# B&R Automation Studio project NAELD004C00R10L518F00 (part 2)

### IoMap.iom - X20CP0483/IoMap.iom
```iecst
VAR_CONFIG
	::DInput:a_bPhysicalDI[1] AT %IX."X20DI9372".DigitalInput01;
	::DInput:a_bPhysicalDI[2] AT %IX."X20DI9372".DigitalInput02;
	::DInput:a_bPhysicalDI[3] AT %IX."X20DI9372".DigitalInput03;
	::DInput:a_bPhysicalDI[4] AT %IX."X20DI9372".DigitalInput04;
	::DInput:a_bPhysicalDI[5] AT %IX."X20DI9372".DigitalInput05;
	::DInput:a_bPhysicalDI[6] AT %IX."X20DI9372".DigitalInput06;
	::DInput:a_bPhysicalDI[7] AT %IX."X20DI9372".DigitalInput07;
	::DInput:a_bPhysicalDI[8] AT %IX."X20DI9372".DigitalInput08;
	::DInput:a_bPhysicalDI[9] AT %IX."X20DI9372".DigitalInput09;
	::DInput:a_bPhysicalDI[10] AT %IX."X20DI9372".DigitalInput10;
	::DInput:a_bPhysicalDI[11] AT %IX."X20DI9372".DigitalInput11;
	::DInput:a_bPhysicalDI[12] AT %IX."X20DI9372".DigitalInput12;
	::DInput:a_bPhysicalDI[13] AT %IX."X20DI9372a".DigitalInput01;
	::DInput:a_bPhysicalDI[14] AT %IX."X20DI9372a".DigitalInput02;
	::DInput:a_bPhysicalDI[15] AT %IX."X20DI9372a".DigitalInput03;
	::DInput:a_bPhysicalDI[16] AT %IX."X20DI9372a".DigitalInput04;
	::DInput:a_bPhysicalDI[17] AT %IX."X20DI9372a".DigitalInput05;
	::DInput:a_bPhysicalDI[18] AT %IX."X20DI9372a".DigitalInput06;
	::DInput:a_bPhysicalDI[19] AT %IX."X20DI9372a".DigitalInput07;
	::DInput:a_bPhysicalDI[20] AT %IX."X20DI9372a".DigitalInput08;
	::DInput:a_bPhysicalDI[21] AT %IX."X20DI9372a".DigitalInput09;
	::DInput:a_bPhysicalDI[22] AT %IX."X20DI9372a".DigitalInput10;
	::DInput:a_bPhysicalDI[23] AT %IX."X20DI9372a".DigitalInput11;
	::DInput:a_bPhysicalDI[24] AT %IX."X20DI9372a".DigitalInput12;
	::DInput:a_bPhysicalDI[25] AT %IX."X20DI9372b".DigitalInput01;
	::DInput:a_bPhysicalDI[26] AT %IX."X20DI9372b".DigitalInput02;
	::DInput:a_bPhysicalDI[27] AT %IX."X20DI9372b".DigitalInput03;
	::DInput:a_bPhysicalDI[28] AT %IX."X20DI9372b".DigitalInput04;
	::DInput:a_bPhysicalDI[29] AT %IX."X20DI9372b".DigitalInput05;
	::DInput:a_bPhysicalDI[30] AT %IX."X20DI9372b".DigitalInput06;
	::DInput:a_bPhysicalDI[31] AT %IX."X20DI9372b".DigitalInput07;
	::DInput:a_bPhysicalDI[32] AT %IX."X20DI9372b".DigitalInput08;
	::DInput:a_bPhysicalDI[33] AT %IX."X20DI9372b".DigitalInput09;
	::DInput:a_bPhysicalDI[34] AT %IX."X20DI9372b".DigitalInput10;
	::DInput:a_bPhysicalDI[35] AT %IX."X20DI9372b".DigitalInput11;
	::DInput:a_bPhysicalDI[36] AT %IX."X20DI9372b".DigitalInput12;
	::DInput:a_bPhysicalDI[37] AT %IX."X20DI9372c".DigitalInput01;
	::DInput:a_bPhysicalDI[38] AT %IX."X20DI9372c".DigitalInput02;
	::DInput:a_bPhysicalDI[39] AT %IX."X20DI9372c".DigitalInput03;
	::DInput:a_bPhysicalDI[40] AT %IX."X20DI9372c".DigitalInput04;
	::DInput:a_bPhysicalDI[41] AT %IX."X20DI9372c".DigitalInput05;
	::DInput:a_bPhysicalDI[42] AT %IX."X20DI9372c".DigitalInput06;
	::DInput:a_bPhysicalDI[43] AT %IX."X20DI9372c".DigitalInput07;
	::DInput:a_bPhysicalDI[44] AT %IX."X20DI9372c".DigitalInput08;
	::DInput:a_bPhysicalDI[45] AT %IX."X20DI9372c".DigitalInput09;
	::DInput:a_bPhysicalDI[46] AT %IX."X20DI9372c".DigitalInput10;
	::DInput:a_bPhysicalDI[47] AT %IX."X20DI9372c".DigitalInput11;
	::DInput:a_bPhysicalDI[48] AT %IX."X20DI9372c".DigitalInput12;
	::DInput:a_bPhysicalDI[49] AT %IX."X20DI9372d".DigitalInput01;
	::DInput:a_bPhysicalDI[50] AT %IX."X20DI9372d".DigitalInput02;
	::DInput:a_bPhysicalDI[51] AT %IX."X20DI9372d".DigitalInput03;
	::DInput:a_bPhysicalDI[52] AT %IX."X20DI9372d".DigitalInput04;
	::DInput:a_bPhysicalDI[53] AT %IX."X20DI9372d".DigitalInput05;
	::DInput:a_bPhysicalDI[54] AT %IX."X20DI9372d".DigitalInput06;
	::DInput:a_bPhysicalDI[55] AT %IX."X20DI9372d".DigitalInput07;
	::DInput:a_bPhysicalDI[56] AT %IX."X20DI9372d".DigitalInput08;
	::DInput:a_bPhysicalDI[57] AT %IX."X20DI9372d".DigitalInput09;
	::DInput:a_bPhysicalDI[58] AT %IX."X20DI9372d".DigitalInput10;
	::DInput:a_bPhysicalDI[59] AT %IX."X20DI9372d".DigitalInput11;
	::DInput:a_bPhysicalDI[60] AT %IX."X20DI9372d".DigitalInput12;
	::DInput:a_bPhysicalDI[61] AT %IX."X20DI9372e".DigitalInput01;
	::DInput:a_bPhysicalDI[62] AT %IX."X20DI9372e".DigitalInput02;
	::DInput:a_bPhysicalDI[63] AT %IX."X20DI9372e".DigitalInput03;
	::DInput:a_bPhysicalDI[64] AT %IX."X20DI9372e".DigitalInput04;
	::DInput:a_bPhysicalDI[65] AT %IX."X20DI9372e".DigitalInput05;
	::DInput:a_bPhysicalDI[66] AT %IX."X20DI9372e".DigitalInput06;
	::DInput:a_bPhysicalDI[67] AT %IX."X20DI9372e".DigitalInput07;
	::DInput:a_bPhysicalDI[68] AT %IX."X20DI9372e".DigitalInput08;
	::DInput:a_bPhysicalDI[69] AT %IX."X20DI9372e".DigitalInput09;
	::DInput:a_bPhysicalDI[70] AT %IX."X20DI9372e".DigitalInput10;
	::DInput:a_bPhysicalDI[71] AT %IX."X20DI9372e".DigitalInput11;
	::DInput:a_bPhysicalDI[72] AT %IX."X20DI9372e".DigitalInput12;
	::DOutput:a_bPhysicalDO[1] AT %QX."X20DO6321".DigitalOutput01;
	::DOutput:a_bPhysicalDO[2] AT %QX."X20DO6321".DigitalOutput02;
	::DOutput:a_bPhysicalDO[3] AT %QX."X20DO6321".DigitalOutput03;
	::DOutput:a_bPhysicalDO[4] AT %QX."X20DO6321".DigitalOutput04;
	::DOutput:a_bPhysicalDO[5] AT %QX."X20DO6321".DigitalOutput05;
	::DOutput:a_bPhysicalDO[6] AT %QX."X20DO6321".DigitalOutput06;
	::DOutput:a_bPhysicalDO[7] AT %QX."X20DO9321".DigitalOutput01;
	::DOutput:a_bPhysicalDO[8] AT %QX."X20DO9321".DigitalOutput02;
	::DOutput:a_bPhysicalDO[9] AT %QX."X20DO9321".DigitalOutput03;
	::DOutput:a_bPhysicalDO[10] AT %QX."X20DO9321".DigitalOutput04;
	::DOutput:a_bPhysicalDO[11] AT %QX."X20DO9321".DigitalOutput05;
	::DOutput:a_bPhysicalDO[12] AT %QX."X20DO9321".DigitalOutput06;
	::DOutput:a_bPhysicalDO[13] AT %QX."X20DO9321".DigitalOutput07;
	::DOutput:a_bPhysicalDO[14] AT %QX."X20DO9321".DigitalOutput08;
	::DOutput:a_bPhysicalDO[15] AT %QX."X20DO9321".DigitalOutput09;
	::DOutput:a_bPhysicalDO[16] AT %QX."X20DO9321".DigitalOutput10;
	::DOutput:a_bPhysicalDO[17] AT %QX."X20DO9321".DigitalOutput11;
	::DOutput:a_bPhysicalDO[18] AT %QX."X20DO9321".DigitalOutput12;
	::DOutput:a_bPhysicalDO[19] AT %QX."X20DO9321a".DigitalOutput01;
	::DOutput:a_bPhysicalDO[20] AT %QX."X20DO9321a".DigitalOutput02;
	::DOutput:a_bPhysicalDO[21] AT %QX."X20DO9321a".DigitalOutput03;
	::DOutput:a_bPhysicalDO[22] AT %QX."X20DO9321a".DigitalOutput04;
	::DOutput:a_bPhysicalDO[23] AT %QX."X20DO9321a".DigitalOutput05;
	::DOutput:a_bPhysicalDO[24] AT %QX."X20DO9321a".DigitalOutput06;
	::DOutput:a_bPhysicalDO[25] AT %QX."X20DO9321a".DigitalOutput07;
	::DOutput:a_bPhysicalDO[26] AT %QX."X20DO9321a".DigitalOutput08;
	::DOutput:a_bPhysicalDO[27] AT %QX."X20DO9321a".DigitalOutput09;
	::DOutput:a_bPhysicalDO[28] AT %QX."X20DO9321a".DigitalOutput10;
	::DOutput:a_bPhysicalDO[29] AT %QX."X20DO9321a".DigitalOutput11;
	::DOutput:a_bPhysicalDO[30] AT %QX."X20DO9321a".DigitalOutput12;
	::DOutput:a_bPhysicalDO[31] AT %QX."X20DO9321b".DigitalOutput01;
	::DOutput:a_bPhysicalDO[32] AT %QX."X20DO9321b".DigitalOutput02;
	::DOutput:a_bPhysicalDO[33] AT %QX."X20DO9321b".DigitalOutput03;
	::DOutput:a_bPhysicalDO[34] AT %QX."X20DO9321b".DigitalOutput04;
	::DOutput:a_bPhysicalDO[35] AT %QX."X20DO9321b".DigitalOutput05;
	::DOutput:a_bPhysicalDO[36] AT %QX."X20DO9321b".DigitalOutput06;
	::DOutput:a_bPhysicalDO[37] AT %QX."X20DO9321b".DigitalOutput07;
	::DOutput:a_bPhysicalDO[38] AT %QX."X20DO9321b".DigitalOutput08;
	::DOutput:a_bPhysicalDO[39] AT %QX."X20DO9321b".DigitalOutput09;
	::DOutput:a_bPhysicalDO[40] AT %QX."X20DO9321b".DigitalOutput10;
	::DOutput:a_bPhysicalDO[41] AT %QX."X20DO9321b".DigitalOutput11;
	::DOutput:a_bPhysicalDO[42] AT %QX."X20DO9321b".DigitalOutput12;
	::DOutput:a_bPhysicalDO[43] AT %QX."X20DO9321c".DigitalOutput01;
	::DOutput:a_bPhysicalDO[44] AT %QX."X20DO9321c".DigitalOutput02;
	::DOutput:a_bPhysicalDO[45] AT %QX."X20DO9321c".DigitalOutput03;
	::DOutput:a_bPhysicalDO[46] AT %QX."X20DO9321c".DigitalOutput04;
	::DOutput:a_bPhysicalDO[47] AT %QX."X20DO9321c".DigitalOutput05;
	::DOutput:a_bPhysicalDO[48] AT %QX."X20DO9321c".DigitalOutput06;
	::DOutput:a_bPhysicalDO[49] AT %QX."X20DO9321c".DigitalOutput07;
	::DOutput:a_bPhysicalDO[50] AT %QX."X20DO9321c".DigitalOutput08;
	::DOutput:a_bPhysicalDO[51] AT %QX."X20DO9321c".DigitalOutput09;
	::DOutput:a_bPhysicalDO[52] AT %QX."X20DO9321c".DigitalOutput10;
	::DOutput:a_bPhysicalDO[53] AT %QX."X20DO9321c".DigitalOutput11;
	::DOutput:a_bPhysicalDO[54] AT %QX."X20DO9321c".DigitalOutput12;
	::LifterBtm:bModuleOK AT %IX."Lifter".ModuleOk;
	::LifterBtm:tyParamInDriver.uiErrCode_603F AT %IW."Lifter".ErrorCode_603F;
	::LifterBtm:tyParamOutDriver.uiCtrlword_6040 AT %QW."Lifter".Controlword_6040;
	::LifterBtm:tyParamInDriver.uiStatword_6041 AT %IW."Lifter".Statusword_6041;
	::LifterBtm:tyParamOutDriver.siModOfOpt_6060 AT %QB."Lifter".ModesOfOperation_6060;
	::LifterBtm:tyParamInDriver.siModOfOptDisp_6061 AT %IB."Lifter".ModesOfOperationDisplay_6061;
	::LifterBtm:tyParamInDriver.diActualPos_6064 AT %ID."Lifter".PositionActualValue_6064;
	::LifterBtm:tyParamOutDriver.diTargetPos_607A AT %QD."Lifter".TargetPosition_607A;
	::LifterBtm:tyParamOutDriver.udiMoveSpd_6081 AT %QD."Lifter".ProfileVelocity_6081;
	::LifterBtm:tyParamOutDriver.siHmMethod_6098 AT %QB."Lifter".HomingMethod_6098;
	::LifterBtm:tyParamInDriver.udiDigitalInputs_60FD AT %ID."Lifter".DigitalInputs_60FD;
	::LifterBtm:tyParamOutDriver.diJogVel_60FF AT %QD."Lifter".TargetVelocity_60FF;
	::Trav:bModuleOK AT %IX."Traverser".ModuleOk;
	::Trav:tyParamInDriver.uiErrCode_603F AT %IW."Traverser".ErrorCode_603F;
	::Trav:tyParamOutDriver.uiCtrlword_6040 AT %QW."Traverser".Controlword_6040;
	::Trav:tyParamInDriver.uiStatword_6041 AT %IW."Traverser".Statusword_6041;
	::Trav:tyParamOutDriver.siModOfOpt_6060 AT %QB."Traverser".ModesOfOperation_6060;
	::Trav:tyParamInDriver.siModOfOptDisp_6061 AT %IB."Traverser".ModesOfOperationDisplay_6061;
	::Trav:tyParamInDriver.diActualPos_6064 AT %ID."Traverser".PositionActualValue_6064;
	::Trav:tyParamOutDriver.diTargetPos_607A AT %QD."Traverser".TargetPosition_607A;
	::Trav:tyParamOutDriver.udiMoveSpd_6081 AT %QD."Traverser".ProfileVelocity_6081;
	::Trav:tyParamOutDriver.siHmMethod_6098 AT %QB."Traverser".HomingMethod_6098;
	::Trav:tyParamInDriver.udiDigitalInputs_60FD AT %ID."Traverser".DigitalInputs_60FD;
	::Trav:tyParamOutDriver.diJogVel_60FF AT %QD."Traverser".TargetVelocity_60FF;
	::AWOpen:bModuleOK AT %IX."AutoWidthConv".ModuleOk;
	::AWOpen:tyParamInDriver.uiErrCode_603F AT %IW."AutoWidthConv".ErrorCode_603F;
	::AWOpen:tyParamInDriver.uiStatword_6041 AT %IW."AutoWidthConv".Statusword_6041;
	::AWOpen:tyParamInDriver.siModOfOptDisp_6061 AT %IB."AutoWidthConv".ModesOfOperationDisplay_6061;
	::AWOpen:tyParamInDriver.diActualPos_6064 AT %ID."AutoWidthConv".PositionActualValue_6064;
	::AWOpen:tyParamInDriver.udiDigitalInputs_60FD AT %ID."AutoWidthConv".DigitalInputs_60FD;
	::AWOpen:tyParamOutDriver.uiCtrlword_6040 AT %QW."AutoWidthConv".Controlword_6040;
	::AWOpen:tyParamOutDriver.siModOfOpt_6060 AT %QB."AutoWidthConv".ModesOfOperation_6060;
	::AWOpen:tyParamOutDriver.diTargetPos_607A AT %QD."AutoWidthConv".TargetPosition_607A;
	::AWOpen:tyParamOutDriver.udiMoveSpd_6081 AT %QD."AutoWidthConv".ProfileVelocity_6081;
	::AWOpen:tyParamOutDriver.siHmMethod_6098 AT %QB."AutoWidthConv".HomingMethod_6098;
	::AWOpen:tyParamOutDriver.diJogVel_60FF AT %QD."AutoWidthConv".TargetVelocity_60FF;
END_VAR
```

## Configuration 3Mag_LD_pneuRot_roller

### Task classes (Cpu.sw)
```
Cyclic#1 (cycle 10000 us, tolerance 10000 us):
  DInput <- DInput.DInput.prg
  DOutput <- DOutput.DOutput.prg
  PneuNoSenS <- (binary)
Cyclic#2 (cycle 20000 us, tolerance 20000 us):
  BarcodeRdr <- USBBarcodeRdr.BarcodeRdr.prg
  PullConv <- Conv.PullConv.prg
  MagConv2Cl <- MagConv.MagConv2Clp1.prg
  MagConv2C1 <- MagConv.MagConv2Clp2.prg
  MagConv2C2 <- MagConv.MagConv2Clp3.prg
  MagConv2C3 <- MagConv.MagConv2Clp4.prg
  MtrPshr <- MtrPshr.MtrPshr.prg
  PullerPush <- CANOpenServo.PullerPusher.PullerPusher.prg
Cyclic#3 (cycle 50000 us, tolerance 50000 us):
  UI <- UI.UI.prg
  Startup <- Startup.Startup.prg
  Time <- Time.Time.prg
  General <- General.General.prg
  UsrFolder <- UsrFolder.UsrFolder.prg
  LibVer <- LibVer.LibVer.prg
  HWInfo <- HWInfo.HWInfo.prg
  TLBuz <- TLBuz.TLBuz.prg
  Alarm <- Alarm.Alarm.prg
  RstErr <- RstErr.RstErr.prg
  ProdRcp <- ProdRcp.ProdRcp.prg
  MpProdRcp <- MpProdRcp.MpProdRcp.prg
  MagRcp <- MagRcp.MagRcp.prg
  McParam <- McParam.McParam.prg
  NtParam <- NtParam.NtParam.prg
  UsrMgmt <- UsrMgmt.UsrMgmt.prg
  Buffer1 <- Buffer.Buffer1.prg
  Buffer2 <- Buffer.Buffer2.prg
  Buffer3 <- Buffer.Buffer3.prg
  Buffer4 <- Buffer.Buffer4.prg
  USSMEMA1 <- SMEMA.USSMEMA1.prg
  USSMEMA2 <- SMEMA.USSMEMA2.prg
  USSMEMA3 <- SMEMA.USSMEMA3.prg
  USSMEMA4 <- SMEMA.USSMEMA4.prg
  DSSMEMA1 <- SMEMA.DSSMEMA1.prg
  DSSMEMA2 <- SMEMA.DSSMEMA2.prg
  DSSMEMA3 <- SMEMA.DSSMEMA3.prg
  DSSMEMA4 <- SMEMA.DSSMEMA4.prg
  DSSMEMAA <- SMEMA.DSSMEMAA.prg
  DSSMEMAB <- SMEMA.DSSMEMAB.prg
  Pneu2SenIn <- Pneu.Pneu2SenInShutter.prg
  Pneu2SenOu <- Pneu.Pneu2SenOutShutter.prg
  Pneu2SenPu <- Pneu.Pneu2SenPuller.prg
  AWOpen <- CANOpenServo.AW.AWOpen.prg
  Trav <- CANOpenServo.Trav.Trav.prg
  LifterBtm <- CANOpenServo.Lifter.LifterBtm.prg
  Hermes <- Hermes.Hermes.prg
  DSHermesA <- Hermes.DSHermesA.prg
  DSHermesB <- Hermes.DSHermesB.prg
  RmtHermes <- Hermes.RmtHermes.prg
  SvyHermes <- Hermes.SvyHermes.prg
  LFLeader <- LF.LFLeader.prg
  LFFollower <- LF.LFFollower.prg
  Follower1 <- LF.Follower1.prg
  Follower2 <- LF.Follower2.prg
  AutoRcp <- AutoRcp.AutoRcp.prg
  LCS <- LCS.LCS.prg
  LCSMngRcp <- LCS.LCSMngRcp.prg
  LCSLF <- LCS.LCSLF.prg
  Ops <- Operations.Ops.prg
  OpsTravLif <- Operations.OpsTravLifLD.prg
  OpsMagConv <- Operations.OpsMagConvLD1.prg
  OpsMagCon1 <- Operations.OpsMagConvLD2.prg
  OpsMagCon2 <- Operations.OpsMagConvLD3.prg
  OpsMagCon3 <- Operations.OpsMagConvLD4.prg
  AGV <- AGVCom.AGV.prg
  AGV1 <- AGVCom.AGV1.prg
  AGV2 <- AGVCom.AGV2.prg
  AGV3 <- AGVCom.AGV3.prg
  AGV4 <- AGVCom.AGV4.prg
  Pneu2SenSe <- Pneu.SelClamp.Pneu2SenSelClamp1.prg
  Pneu2SenS1 <- Pneu.SelClamp.Pneu2SenSelClamp2.prg
  Pneu2SenS2 <- Pneu.SelClamp.Pneu2SenSelClamp3.prg
  Pneu2SenS3 <- Pneu.SelClamp.Pneu2SenSelClamp4.prg
  Simu <- Simulation.Simu.prg
  USSOT1 <- SOT.USSOT1.prg
  DSSOT1 <- SOT.DSSOT1.prg
  USSOT2 <- SOT.USSOT2.prg
  DSSOT2 <- SOT.DSSOT2.prg
  USSOT3 <- SOT.USSOT3.prg
  DSSOT3 <- SOT.DSSOT3.prg
  USSOT4 <- SOT.USSOT4.prg
  DSSOT4 <- SOT.DSSOT4.prg
  Machine <- Machine.Machine.prg
  MagRcp2 <- MagRcp.MagRcp1.prg
  Pneu2SenMa <- Pneu.MagSafetyBar.Pneu2SenMag1SafetyBar.prg
  Pneu2SenM1 <- Pneu.MagSafetyBar.Pneu2SenMag2SafetyBar.prg
  Pneu2SenM2 <- Pneu.MagSafetyBar.Pneu2SenMag3SafetyBar.prg
  Pneu2SenM3 <- Pneu.MagSafetyBar.Pneu2SenMag4SafetyBar.prg
  Pneu2SenI2 <- Pneu.Pneu2SenInShutter2.prg
  Pneu2SenI3 <- Pneu.Pneu2SenInShutter3.prg
  AWPushOrPu <- CANOpenServo.AW.AWPushOrPuller.prg
  OpsLifMagL <- Operations.OpsLifMagLD.prg
  Machine2 <- Machine.Machine1.prg
  Frame <- RS232.DVFrame.Frame.prg
DataObjects: Acp10sys
VcDataObjects: Visu <- UI.Visu.dob
Binaries: vccdt, vccbmp, Visu03, vcfile, arial, vctcal, arialxsr, vcmgr, visvc, vccstr, vcbclass, vccbtn, vcgclass, vcdsint, vcnet, vccline, vcshared, vccddbox, arialbd, vccnum, vcpdvnc, vcpdsw, vccslider, vccbar, vcctext, Visu01, arialbi, vcfntttf, vccovl, vccshape, vcalarm, Visu02, vcrt, udbdef, vccpopup, vcdsloc, vcchspot, TCData, vcpfgen, vccalarm, arsvcreg, User, sysconf, ashwac, ashwd, Role, asfw, arconfig, iomap, Config, vcpfar00, acp10cfg, Acp10map, vcpkat, OpcUaMap
Libraries: standard, runtime, astime, asstring, operator, AsIecCon, AsCANopen, visapi, FileIO, AsIODiag, AsMem, dvframe, AsOpcUac, AsARCfg, sys_lib, AsTCP, MpRecipe, AsFltGen, brsystem, NtBuffer, NtConv, NtFileIO, NtLogFile, NtMem, NtMessage, NtOPCUA, NtOvenInfo, NtPneu, NtRS232, NtTLBuz, NtTCP, NtVersion, MpCom, MpBase, AsUSB, NtSMEMA, NtSOT, NtGeneral, NtUI, NtUSB, NtLF, NtRecipe, NtMotion, NtHermes, sprintf, AsMath, vcresman, dataobj, powerlnk
```

### Hardware
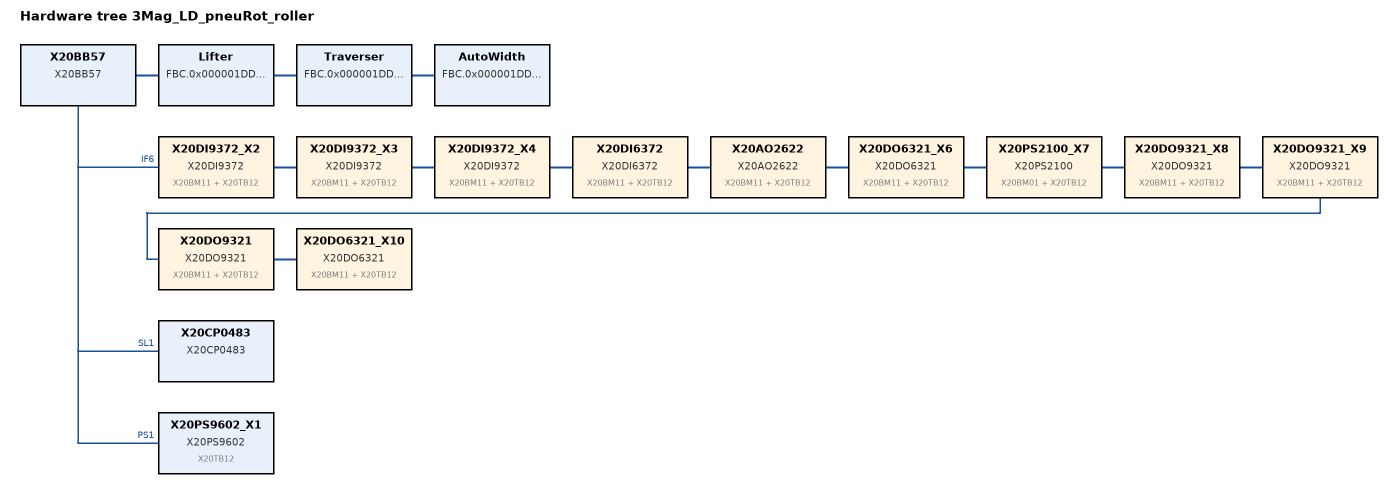
```
AutoWidth : FBC.0x000001DD.0x00000001.NUTEK_DELTA_EDS_V101 v1.0 (OrderNumber=NUTEK_DELTA_V101)  [CAN1 -> Traverser.CAN2 (NodeNumber=16)]
Lifter : FBC.0x000001DD.0x00000001.NUTEK_DELTA_EDS_V101 v1.0 (OrderNumber=NUTEK_DELTA_V101)  [CAN1 -> X20BB57.IF7 (NodeNumber=17)]
Traverser : FBC.0x000001DD.0x00000001.NUTEK_DELTA_EDS_V101 v1.0 (OrderNumber=NUTEK_DELTA_V101)  [CAN1 -> Lifter.CAN2]
X20AO2622 : X20AO2622 v1.2.0.0  [SS1 -> X20TB12l.SS; SL -> X20BM11j.SL1]
X20BB57 : X20BB57 v1.1.1.0
  Connector IF1:
    Baudrate = 9600
    Parity = N
  Connector IF7:
    Baudrate = 1000000
    ActivateCanOpen = 1
    p100c_parametervalue = 1000
    p100d_parametervalue = 3
X20BM01 : X20BM01 v2.1.0.0  [X2X1 -> X20BM11d.X2X2]
X20BM11 : X20BM11 v1.0.0.1  [X2X1 -> X20BB57.IF6]
X20BM11a : X20BM11 v1.0.0.1  [X2X1 -> X20BM11.X2X2]
X20BM11b : X20BM11 v1.0.0.1  [X2X1 -> X20BM11a.X2X2]
X20BM11d : X20BM11 v1.0.0.1  [X2X1 -> X20BM11j.X2X2]
X20BM11e : X20BM11 v1.0.0.1  [X2X1 -> X20BM01.X2X2]
X20BM11f : X20BM11 v1.0.0.1  [X2X1 -> X20BM11e.X2X2]
X20BM11g : X20BM11 v1.0.0.1  [X2X1 -> X20BM11i.X2X2]
X20BM11h : X20BM11 v1.0.0.1  [X2X1 -> X20BM11b.X2X2]
X20BM11i : X20BM11 v1.0.0.1  [X2X1 -> X20BM11f.X2X2]
X20BM11j : X20BM11 v1.0.0.1  [X2X1 -> X20BM11h.X2X2]
X20CP0483 : X20CP0483 v1.2.1.0  [SL -> X20BB57.SL1]
  Connector IF2:
    ActivateDevice = 1
    Mode = Manual
    InternetAddress = 172.22.84.32
    SubnetMask = 255.255.0.0
    Vnc1
    VncVcObjectName1 = Visu
    VncKeyMappingFile1 = 
    VncMaxConnections1 = 3
    VncRefreshRate1 = 100
    ActivateSnmp = 2
  ConfigurationID = NAELD004
  UserPartitionSize = 150
  VolatileGlobalPvSize = 80000
  EnableUsbRemoteInstall = 1
  TimerDeviceType = SWIOTIMER
  Cyclic1Duration = 10000
  Cyclic1Tolerance = 10000
  Cyclic2Duration = 20000
  Cyclic2Tolerance = 20000
  Cyclic3Duration = 50000
  Cyclic3Tolerance = 50000
  Cyclic4Duration = 10000
  Cyclic4Tolerance = 10000
  Cyclic5Duration = 200000
  Cyclic5Tolerance = 200000
  Cyclic6Duration = 500000
  Cyclic6Tolerance = 500000
  Cyclic7Duration = 1000000
  Cyclic7Tolerance = 1000000
  Cyclic8Duration = 10000
  Cyclic8Tolerance = 10000
  FileDevice1
  FileDeviceName1 = F
  FileDevicePath1 = F:
  FileDevice2
  FileDeviceName2 = User
  FileDevicePath2 = F:\User
  FileDevice3
  FileDeviceName3 = Private
  FileDevicePath3 = F:\Private
  FileDevice4
  FileDeviceName4 = CustomerUser
  FileDevicePath4 = F:\User\UserMgmt
  FileDevice5
  FileDeviceName5 = ProdRcp
  FileDevicePath5 = F:\User\ProductRecipe
  FileDevice6
  FileDeviceName6 = MagRcp
  FileDevicePath6 = F:\User\MagazineRecipe
  FileDevice7
  FileDeviceName7 = Alarm
  FileDevicePath7 = F:\User\Alarm
  FileDevice8
  FileDeviceName8 = McParam
  FileDevicePath8 = F:\User\MachineParameter
  FileDevice9
  FileDeviceName9 = NtParam
  FileDevicePath9 = F:\Private\NutekParameter
  FileDevice10
  FileDeviceName10 = LibVer
  FileDevicePath10 = F:\User\LibrariesVersion
  FileDevice11
  FileDeviceName11 = Retain
  FileDevicePath11 = F:\User\Retain
  FileDevice12
  FileDeviceName12 = Log
  FileDevicePath12 = F:\User\Log
  FileDevice13
  FileDeviceName13 = LCS
  FileDevicePath13 = F:\User\LCS
  FileDevice14
  FileDeviceName14 = MpProdRcp
  FileDevicePath14 = F:\User\ProductRecipeXml
  FileDevice15
  FileDeviceName15 = MpNtParam
  FileDevicePath15 = F:\Private\NutekParameterXml
  FtpUser1
  FtpUsername1 = NTAFTP
  FtpUserPassword1 = JmcONQZEIGyG0Pt+VekJRbxmc4fxS8REPwlCJguEtEY=  // NTA4BH
  FtpUserSalt1 = smKszLJT
  FTPAccessRight1 = 0
  FTPdevice1 = ALL
  FtpUser2
  FtpUsername2 = admin
  FtpUserPassword2 = GulCMI/jV0v16Ew6MS+jrzqmTLk+NRkNo3Y+jAhzSzY=  // admin
  FtpUserSalt2 = robUzvv7
  FTPAccessRight2 = 0
  FTPMSPartition2 = SYSTEM
  FTPMSpath2 = User
  FtpUser3
  FtpUsername3 = LCS
  FtpUserPassword3 = 6XI8rzr3QlcLzq1fKGxRBMxxRW19t00F0QlEDJIXmLc=  // LCS
  FtpUserSalt3 = Xz6TWjSu
  FTPMSPartition3 = SYSTEM
  FTPMSpath3 = User\LCS
  ActivateOpcUa = 1
  OpcUa_ConversationSecurityPolicy_EnableBasic256Rsa256 = 0
  OpcUaInformationModels_PV_Version = 1
X20DI6372 : X20DI6372 v1.1.0.0  [SS1 -> X20TB12j.SS; SL -> X20BM11h.SL1]
X20DI9372_X2 : X20DI9372 v1.1.0.0  [SS1 -> X20TB12a.SS; SL -> X20BM11.SL1]
  Supervision = off
X20DI9372_X3 : X20DI9372 v1.1.0.0  [SS1 -> X20TB12b.SS; SL -> X20BM11a.SL1]
  Supervision = off
X20DI9372_X4 : X20DI9372 v1.1.0.0  [SS1 -> X20TB12c.SS; SL -> X20BM11b.SL1]
  Supervision = off
X20DO6321_X10 : X20DO6321 v1.1.0.0  [SS1 -> X20TB12i.SS; SL -> X20BM11g.SL1]
X20DO6321_X6 : X20DO6321 v1.1.0.0  [SS1 -> X20TB12e.SS; SL -> X20BM11d.SL1]
  Supervision = off
X20DO9321 : X20DO9321 v1.1.0.0  [SS1 -> X20TB12k.SS; SL -> X20BM11i.SL1]
X20DO9321_X8 : X20DO9321 v1.1.0.0  [SS1 -> X20TB12g.SS; SL -> X20BM11e.SL1]
  Supervision = off
X20DO9321_X9 : X20DO9321 v1.1.0.0  [SS1 -> X20TB12h.SS; SL -> X20BM11f.SL1]
  Supervision = off
X20PS2100_X7 : X20PS2100 v1.2.0.0  [SS1 -> X20TB12f.SS; SL -> X20BM01.SL1]
  Supervision = off
X20PS9602_X1 : X20PS9602 v1.0.2.0  [PS -> X20BB57.PS1; SS1 -> X20TB12.SS]
X20TB12 : X20TB12 v1.0.0.0
X20TB12a : X20TB12 v1.0.0.0
X20TB12b : X20TB12 v1.0.0.0
X20TB12c : X20TB12 v1.0.0.0
X20TB12e : X20TB12 v1.0.0.0
X20TB12f : X20TB12 v1.0.0.0
X20TB12g : X20TB12 v1.0.0.0
X20TB12h : X20TB12 v1.0.0.0
X20TB12i : X20TB12 v1.0.0.0
X20TB12j : X20TB12 v1.0.0.0
X20TB12k : X20TB12 v1.0.0.0
X20TB12l : X20TB12 v1.0.0.0
```

### IoMap.iom - X20CP0483/IoMap.iom
```iecst
VAR_CONFIG
	::DInput:a_bPhysicalDI[1] AT %IX."X20DI9372_X2".DigitalInput01;
	::DInput:a_bPhysicalDI[2] AT %IX."X20DI9372_X2".DigitalInput02;
	::DInput:a_bPhysicalDI[3] AT %IX."X20DI9372_X2".DigitalInput03;
	::DInput:a_bPhysicalDI[4] AT %IX."X20DI9372_X2".DigitalInput04;
	::DInput:a_bPhysicalDI[5] AT %IX."X20DI9372_X2".DigitalInput05;
	::DInput:a_bPhysicalDI[6] AT %IX."X20DI9372_X2".DigitalInput06;
	::DInput:a_bPhysicalDI[7] AT %IX."X20DI9372_X2".DigitalInput07;
	::DInput:a_bPhysicalDI[8] AT %IX."X20DI9372_X2".DigitalInput08;
	::DInput:a_bPhysicalDI[9] AT %IX."X20DI9372_X2".DigitalInput09;
	::DInput:a_bPhysicalDI[10] AT %IX."X20DI9372_X2".DigitalInput10;
	::DInput:a_bPhysicalDI[11] AT %IX."X20DI9372_X2".DigitalInput11;
	::DInput:a_bPhysicalDI[12] AT %IX."X20DI9372_X2".DigitalInput12;
	::DInput:a_bPhysicalDI[13] AT %IX."X20DI9372_X3".DigitalInput01;
	::DInput:a_bPhysicalDI[14] AT %IX."X20DI9372_X3".DigitalInput02;
	::DInput:a_bPhysicalDI[15] AT %IX."X20DI9372_X3".DigitalInput03;
	::DInput:a_bPhysicalDI[16] AT %IX."X20DI9372_X3".DigitalInput04;
	::DInput:a_bPhysicalDI[17] AT %IX."X20DI9372_X3".DigitalInput05;
	::DInput:a_bPhysicalDI[18] AT %IX."X20DI9372_X3".DigitalInput06;
	::DInput:a_bPhysicalDI[19] AT %IX."X20DI9372_X3".DigitalInput07;
	::DInput:a_bPhysicalDI[20] AT %IX."X20DI9372_X3".DigitalInput08;
	::DInput:a_bPhysicalDI[21] AT %IX."X20DI9372_X3".DigitalInput09;
	::DInput:a_bPhysicalDI[22] AT %IX."X20DI9372_X3".DigitalInput10;
	::DInput:a_bPhysicalDI[23] AT %IX."X20DI9372_X3".DigitalInput11;
	::DInput:a_bPhysicalDI[24] AT %IX."X20DI9372_X3".DigitalInput12;
	::DInput:a_bPhysicalDI[25] AT %IX."X20DI9372_X4".DigitalInput01;
	::DInput:a_bPhysicalDI[26] AT %IX."X20DI9372_X4".DigitalInput02;
	::DInput:a_bPhysicalDI[27] AT %IX."X20DI9372_X4".DigitalInput03;
	::DInput:a_bPhysicalDI[28] AT %IX."X20DI9372_X4".DigitalInput04;
	::DInput:a_bPhysicalDI[29] AT %IX."X20DI9372_X4".DigitalInput05;
	::DInput:a_bPhysicalDI[30] AT %IX."X20DI9372_X4".DigitalInput06;
	::DInput:a_bPhysicalDI[31] AT %IX."X20DI9372_X4".DigitalInput07;
	::DInput:a_bPhysicalDI[32] AT %IX."X20DI9372_X4".DigitalInput08;
	::DInput:a_bPhysicalDI[33] AT %IX."X20DI9372_X4".DigitalInput09;
	::DInput:a_bPhysicalDI[34] AT %IX."X20DI9372_X4".DigitalInput10;
	::DInput:a_bPhysicalDI[35] AT %IX."X20DI9372_X4".DigitalInput11;
	::DInput:a_bPhysicalDI[36] AT %IX."X20DI9372_X4".DigitalInput12;
	::DOutput:a_bPhysicalDO[1] AT %QX."X20DO6321_X6".DigitalOutput01;
	::DOutput:a_bPhysicalDO[2] AT %QX."X20DO6321_X6".DigitalOutput02;
	::DOutput:a_bPhysicalDO[3] AT %QX."X20DO6321_X6".DigitalOutput03;
	::DOutput:a_bPhysicalDO[4] AT %QX."X20DO6321_X6".DigitalOutput04;
	::DOutput:a_bPhysicalDO[5] AT %QX."X20DO6321_X6".DigitalOutput05;
	::DOutput:a_bPhysicalDO[6] AT %QX."X20DO6321_X6".DigitalOutput06;
	::DOutput:a_bPhysicalDO[7] AT %QX."X20DO9321_X8".DigitalOutput01;
	::DOutput:a_bPhysicalDO[8] AT %QX."X20DO9321_X8".DigitalOutput02;
	::DOutput:a_bPhysicalDO[9] AT %QX."X20DO9321_X8".DigitalOutput03;
	::DOutput:a_bPhysicalDO[10] AT %QX."X20DO9321_X8".DigitalOutput04;
	::DOutput:a_bPhysicalDO[11] AT %QX."X20DO9321_X8".DigitalOutput05;
	::DOutput:a_bPhysicalDO[12] AT %QX."X20DO9321_X8".DigitalOutput06;
	::DOutput:a_bPhysicalDO[13] AT %QX."X20DO9321_X8".DigitalOutput07;
	::DOutput:a_bPhysicalDO[14] AT %QX."X20DO9321_X8".DigitalOutput08;
	::DOutput:a_bPhysicalDO[15] AT %QX."X20DO9321_X8".DigitalOutput09;
	::DOutput:a_bPhysicalDO[16] AT %QX."X20DO9321_X8".DigitalOutput10;
	::DOutput:a_bPhysicalDO[17] AT %QX."X20DO9321_X8".DigitalOutput11;
	::DOutput:a_bPhysicalDO[18] AT %QX."X20DO9321_X8".DigitalOutput12;
	::DOutput:a_bPhysicalDO[19] AT %QX."X20DO9321_X9".DigitalOutput01;
	::DOutput:a_bPhysicalDO[20] AT %QX."X20DO9321_X9".DigitalOutput02;
	::DOutput:a_bPhysicalDO[21] AT %QX."X20DO9321_X9".DigitalOutput03;
	::DOutput:a_bPhysicalDO[22] AT %QX."X20DO9321_X9".DigitalOutput04;
	::DOutput:a_bPhysicalDO[23] AT %QX."X20DO9321_X9".DigitalOutput05;
	::DOutput:a_bPhysicalDO[24] AT %QX."X20DO9321_X9".DigitalOutput06;
	::AWOpen:bModuleOK AT %IX."AutoWidth".ModuleOk;
	::AWOpen:tyParamInDriver.uiErrCode_603F AT %IW."AutoWidth".ErrorCode_603F;
	::AWOpen:tyParamOutDriver.uiCtrlword_6040 AT %QW."AutoWidth".Controlword_6040;
	::AWOpen:tyParamInDriver.uiStatword_6041 AT %IW."AutoWidth".Statusword_6041;
	::AWOpen:tyParamOutDriver.siModOfOpt_6060 AT %QB."AutoWidth".ModesOfOperation_6060;
	::AWOpen:tyParamInDriver.siModOfOptDisp_6061 AT %IB."AutoWidth".ModesOfOperationDisplay_6061;
	::AWOpen:tyParamInDriver.diActualPos_6064 AT %ID."AutoWidth".PositionActualValue_6064;
	::AWOpen:tyParamOutDriver.diTargetPos_607A AT %QD."AutoWidth".TargetPosition_607A;
	::AWOpen:tyParamOutDriver.udiMoveSpd_6081 AT %QD."AutoWidth".ProfileVelocity_6081;
	::AWOpen:tyParamOutDriver.siHmMethod_6098 AT %QB."AutoWidth".HomingMethod_6098;
	::AWOpen:tyParamInDriver.udiDigitalInputs_60FD AT %ID."AutoWidth".DigitalInputs_60FD;
	::AWOpen:tyParamOutDriver.diJogVel_60FF AT %QD."AutoWidth".TargetVelocity_60FF;
	::LifterBtm:bModuleOK AT %IX."Lifter".ModuleOk;
	::LifterBtm:tyParamInDriver.uiErrCode_603F AT %IW."Lifter".ErrorCode_603F;
	::LifterBtm:tyParamOutDriver.uiCtrlword_6040 AT %QW."Lifter".Controlword_6040;
	::LifterBtm:tyParamInDriver.uiStatword_6041 AT %IW."Lifter".Statusword_6041;
	::LifterBtm:tyParamOutDriver.siModOfOpt_6060 AT %QB."Lifter".ModesOfOperation_6060;
	::LifterBtm:tyParamInDriver.siModOfOptDisp_6061 AT %IB."Lifter".ModesOfOperationDisplay_6061;
	::LifterBtm:tyParamInDriver.diActualPos_6064 AT %ID."Lifter".PositionActualValue_6064;
	::LifterBtm:tyParamOutDriver.diTargetPos_607A AT %QD."Lifter".TargetPosition_607A;
	::LifterBtm:tyParamOutDriver.udiMoveSpd_6081 AT %QD."Lifter".ProfileVelocity_6081;
	::LifterBtm:tyParamOutDriver.siHmMethod_6098 AT %QB."Lifter".HomingMethod_6098;
	::LifterBtm:tyParamInDriver.udiDigitalInputs_60FD AT %ID."Lifter".DigitalInputs_60FD;
	::LifterBtm:tyParamOutDriver.diJogVel_60FF AT %QD."Lifter".TargetVelocity_60FF;
	::Trav:bModuleOK AT %IX."Traverser".ModuleOk;
	::Trav:tyParamInDriver.uiErrCode_603F AT %IW."Traverser".ErrorCode_603F;
	::Trav:tyParamOutDriver.uiCtrlword_6040 AT %QW."Traverser".Controlword_6040;
	::Trav:tyParamInDriver.uiStatword_6041 AT %IW."Traverser".Statusword_6041;
	::Trav:tyParamOutDriver.siModOfOpt_6060 AT %QB."Traverser".ModesOfOperation_6060;
	::Trav:tyParamInDriver.siModOfOptDisp_6061 AT %IB."Traverser".ModesOfOperationDisplay_6061;
	::Trav:tyParamInDriver.diActualPos_6064 AT %ID."Traverser".PositionActualValue_6064;
	::Trav:tyParamOutDriver.diTargetPos_607A AT %QD."Traverser".TargetPosition_607A;
	::Trav:tyParamOutDriver.udiMoveSpd_6081 AT %QD."Traverser".ProfileVelocity_6081;
	::Trav:tyParamOutDriver.siHmMethod_6098 AT %QB."Traverser".HomingMethod_6098;
	::Trav:tyParamInDriver.udiDigitalInputs_60FD AT %ID."Traverser".DigitalInputs_60FD;
	::Trav:tyParamOutDriver.diJogVel_60FF AT %QD."Traverser".TargetVelocity_60FF;
	::DOutput:a_bPhysicalDO[25] AT %QX."X20DO9321_X9".DigitalOutput07;
	::DOutput:a_bPhysicalDO[26] AT %QX."X20DO9321_X9".DigitalOutput08;
	::DOutput:a_bPhysicalDO[27] AT %QX."X20DO9321_X9".DigitalOutput09;
	::DOutput:a_bPhysicalDO[28] AT %QX."X20DO9321_X9".DigitalOutput10;
	::DOutput:a_bPhysicalDO[29] AT %QX."X20DO9321_X9".DigitalOutput11;
	::DOutput:a_bPhysicalDO[30] AT %QX."X20DO9321_X9".DigitalOutput12;
	::DOutput:a_bPhysicalDO[43] AT %QX."X20DO6321_X10".DigitalOutput01;
	::DOutput:a_bPhysicalDO[44] AT %QX."X20DO6321_X10".DigitalOutput02;
	::DOutput:a_bPhysicalDO[45] AT %QX."X20DO6321_X10".DigitalOutput03;
	::DOutput:a_bPhysicalDO[46] AT %QX."X20DO6321_X10".DigitalOutput04;
	::DOutput:a_bPhysicalDO[47] AT %QX."X20DO6321_X10".DigitalOutput05;
	::DOutput:a_bPhysicalDO[48] AT %QX."X20DO6321_X10".DigitalOutput06;
	::DInput:a_bPhysicalDI[49] AT %IX."X20DI6372".DigitalInput01;
	::DInput:a_bPhysicalDI[50] AT %IX."X20DI6372".DigitalInput02;
	::DInput:a_bPhysicalDI[51] AT %IX."X20DI6372".DigitalInput03;
	::DInput:a_bPhysicalDI[52] AT %IX."X20DI6372".DigitalInput04;
	::DInput:a_bPhysicalDI[53] AT %IX."X20DI6372".DigitalInput05;
	::DInput:a_bPhysicalDI[54] AT %IX."X20DI6372".DigitalInput06;
	::DOutput:a_bPhysicalDO[31] AT %QX."X20DO9321".DigitalOutput01;
	::DOutput:a_bPhysicalDO[32] AT %QX."X20DO9321".DigitalOutput02;
	::DOutput:a_bPhysicalDO[33] AT %QX."X20DO9321".DigitalOutput03;
	::DOutput:a_bPhysicalDO[34] AT %QX."X20DO9321".DigitalOutput04;
	::DOutput:a_bPhysicalDO[35] AT %QX."X20DO9321".DigitalOutput05;
	::DOutput:a_bPhysicalDO[36] AT %QX."X20DO9321".DigitalOutput06;
	::DOutput:a_bPhysicalDO[37] AT %QX."X20DO9321".DigitalOutput07;
	::DOutput:a_bPhysicalDO[38] AT %QX."X20DO9321".DigitalOutput08;
	::DOutput:a_bPhysicalDO[40] AT %QX."X20DO9321".DigitalOutput10;
	::DOutput:a_bPhysicalDO[41] AT %QX."X20DO9321".DigitalOutput11;
	::DOutput:a_bPhysicalDO[42] AT %QX."X20DO9321".DigitalOutput12;
	::DOutput:a_bPhysicalDO[39] AT %QX."X20DO9321".DigitalOutput09;
	::MtrPshr:iAnalogTorque AT %QW."X20AO2622".AnalogOutput01;
END_VAR
```

## Configuration 3Mag_RotMtrPuller_Del_NoRoller

CPU X20CP0483, AutomationRuntime B4.82, Build 4.1.2, Safety 0.0, Vc V4.72.1

### Task classes (Cpu.sw)
```
Cyclic#1 (cycle 10000 us, tolerance 10000 us):
  DInput <- DInput.DInput.prg
  DOutput <- DOutput.DOutput.prg
Cyclic#2 (cycle 20000 us, tolerance 20000 us):
  BarcodeRdr <- USBBarcodeRdr.BarcodeRdr.prg
  PullConv <- Conv.PullConv.prg
  MagConv2Cl <- MagConv.MagConv2Clp1.prg
  MagConv2C2 <- MagConv.MagConv2Clp3.prg
  MagConv2C3 <- MagConv.MagConv2Clp4.prg
  MagConv2C1 <- MagConv.MagConv2Clp2.prg
  MtrPshr <- MtrPshr.MtrPshr.prg
  PullerPush <- CANOpenServo.PullerPusher.PullerPusher.prg
Cyclic#3 (cycle 50000 us, tolerance 50000 us):
  UI <- UI.UI.prg
  Startup <- Startup.Startup.prg
  General <- General.General.prg
  UsrFolder <- UsrFolder.UsrFolder.prg
  LibVer <- LibVer.LibVer.prg
  Time <- Time.Time.prg
  HWInfo <- HWInfo.HWInfo.prg
  TLBuz <- TLBuz.TLBuz.prg
  Alarm <- Alarm.Alarm.prg
  RstErr <- RstErr.RstErr.prg
  ProdRcp <- ProdRcp.ProdRcp.prg
  MpProdRcp <- MpProdRcp.MpProdRcp.prg
  MagRcp <- MagRcp.MagRcp.prg
  MagRcp1 <- MagRcp.MagRcp1.prg
  McParam <- McParam.McParam.prg
  NtParam <- NtParam.NtParam.prg
  UsrMgmt <- UsrMgmt.UsrMgmt.prg
  Buffer1 <- Buffer.Buffer1.prg
  Buffer2 <- Buffer.Buffer2.prg
  Buffer3 <- Buffer.Buffer3.prg
  Buffer4 <- Buffer.Buffer4.prg
  USSMEMA1 <- SMEMA.USSMEMA1.prg
  USSMEMA2 <- SMEMA.USSMEMA2.prg
  USSMEMA3 <- SMEMA.USSMEMA3.prg
  USSMEMA4 <- SMEMA.USSMEMA4.prg
  DSSMEMA1 <- SMEMA.DSSMEMA1.prg
  DSSMEMA2 <- SMEMA.DSSMEMA2.prg
  DSSMEMA3 <- SMEMA.DSSMEMA3.prg
  DSSMEMA4 <- SMEMA.DSSMEMA4.prg
  DSSMEMAA <- SMEMA.DSSMEMAA.prg
  DSSMEMAB <- SMEMA.DSSMEMAB.prg
  Pneu2SenIn <- Pneu.Pneu2SenInShutter.prg
  Pneu2SenOu <- Pneu.Pneu2SenOutShutter.prg
  Pneu2SenPu <- Pneu.Pneu2SenPuller.prg
  Pneu2SenI1 <- Pneu.Pneu2SenInShutter2.prg
  Pneu2SenI2 <- Pneu.Pneu2SenInShutter3.prg
  Pneu2SenMa <- Pneu.MagSafetyBar.Pneu2SenMag1SafetyBar.prg
  Pneu2SenM1 <- Pneu.MagSafetyBar.Pneu2SenMag2SafetyBar.prg
  Pneu2SenM2 <- Pneu.MagSafetyBar.Pneu2SenMag3SafetyBar.prg
  Pneu2SenM3 <- Pneu.MagSafetyBar.Pneu2SenMag4SafetyBar.prg
  AWPushOrPu <- CANOpenServo.AW.AWPushOrPuller.prg
  AWOpen <- CANOpenServo.AW.AWOpen.prg
  Trav <- CANOpenServo.Trav.Trav.prg
  LifterBtm <- CANOpenServo.Lifter.LifterBtm.prg
  Hermes <- Hermes.Hermes.prg
  DSHermesA <- Hermes.DSHermesA.prg
  DSHermesB <- Hermes.DSHermesB.prg
  RmtHermes <- Hermes.RmtHermes.prg
  LFLeader <- LF.LFLeader.prg
  LFFollower <- LF.LFFollower.prg
  Follower1 <- LF.Follower1.prg
  Follower2 <- LF.Follower2.prg
  LCS <- LCS.LCS.prg
  LCSMngRcp <- LCS.LCSMngRcp.prg
  LCSLF <- LCS.LCSLF.prg
  Ops <- Operations.Ops.prg
  OpsTravLif <- Operations.OpsTravLifLD.prg
  OpsMagConv <- Operations.OpsMagConvLD1.prg
  OpsMagCon1 <- Operations.OpsMagConvLD2.prg
  OpsMagCon2 <- Operations.OpsMagConvLD3.prg
  OpsMagCon3 <- Operations.OpsMagConvLD4.prg
  OpsLifMagL <- Operations.OpsLifMagLD.prg
  AGV <- AGVCom.AGV.prg
  AGV1 <- AGVCom.AGV1.prg
  AGV2 <- AGVCom.AGV2.prg
  AGV3 <- AGVCom.AGV3.prg
  AGV4 <- AGVCom.AGV4.prg
  Pneu2SenSe <- Pneu.SelClamp.Pneu2SenSelClamp1.prg
  Pneu2SenS1 <- Pneu.SelClamp.Pneu2SenSelClamp2.prg
  Pneu2SenS2 <- Pneu.SelClamp.Pneu2SenSelClamp3.prg
  Pneu2SenS3 <- Pneu.SelClamp.Pneu2SenSelClamp4.prg
  Simu <- Simulation.Simu.prg
  USSOT1 <- SOT.USSOT1.prg
  DSSOT1 <- SOT.DSSOT1.prg
  USSOT2 <- SOT.USSOT2.prg
  DSSOT2 <- SOT.DSSOT2.prg
  USSOT3 <- SOT.USSOT3.prg
  DSSOT3 <- SOT.DSSOT3.prg
  USSOT4 <- SOT.USSOT4.prg
  DSSOT4 <- SOT.DSSOT4.prg
  Machine <- Machine.Machine.prg
  Machine1 <- Machine.Machine1.prg
  Frame <- RS232.DVFrame.Frame.prg
DataObjects: Acp10sys
VcDataObjects: Visu <- UI.Visu.dob
Binaries: vccdt, vccbmp, Visu03, vcfile, arial, vctcal, arialxsr, vcmgr, visvc, vccstr, vcbclass, vccbtn, vcgclass, vcdsint, vcnet, vccline, vcshared, vccddbox, arialbd, vccnum, vcpdvnc, vcpdsw, vccslider, vccbar, vcctext, Visu01, arialbi, vcfntttf, vccovl, vccshape, vcalarm, Visu02, vcrt, udbdef, vccpopup, vcdsloc, vcchspot, TCData, vcpkat, vcpfgen, vccalarm, User, sysconf, ashwac, ashwd, Role, asfw, arconfig, iomap, Config, arsvcreg, acp10cfg, Acp10map, OpcUaMap, vcpfar00
Libraries: standard, runtime, NtLF, astime, asstring, operator, AsIecCon, AsCANopen, visapi, FileIO, AsIODiag, AsMem, dvframe, AsOpcUac, AsARCfg, sys_lib, AsTCP, MpRecipe, AsFltGen, brsystem, NtBuffer, NtConv, NtFileIO, NtLogFile, NtSMEMA, NtMem, NtMessage, NtOPCUA, NtOvenInfo, NtPneu, NtRS232, NtTLBuz, NtTCP, NtVersion, MpCom, MpBase, AsUSB, NtSOT, NtUSB, NtRecipe, NtGeneral, NtUI, NtMotion, vcresman, sprintf, dataobj, powerlnk
```

### Hardware
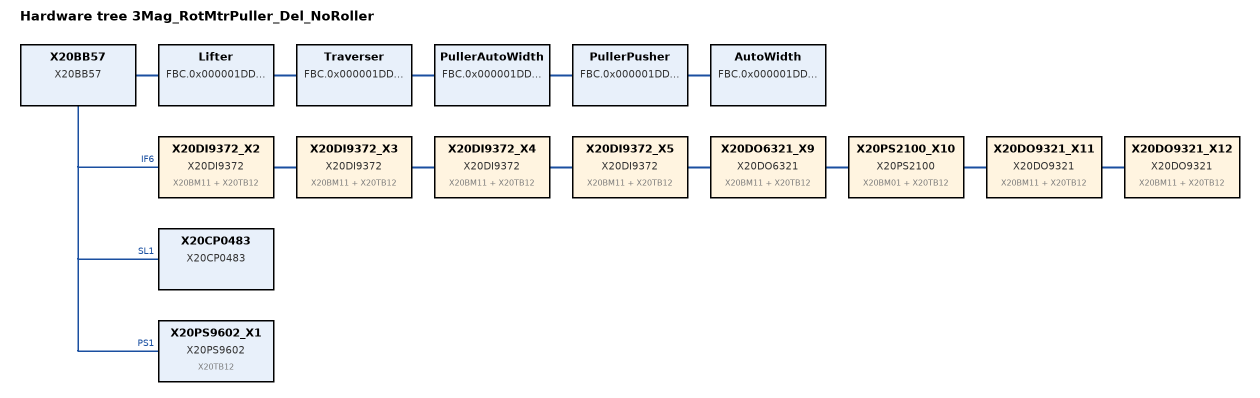
```
AutoWidth : FBC.0x000001DD.0x00000001.NUTEK_DELTA_EDS_V101 v1.0 (OrderNumber=NUTEK_DELTA_V101)  [CAN1 -> PullerPusher.CAN2 (NodeNumber=16)]
Lifter : FBC.0x000001DD.0x00000001.NUTEK_DELTA_EDS_V101 v1.0 (OrderNumber=NUTEK_DELTA_V101)  [CAN1 -> X20BB57.IF7 (NodeNumber=17)]
PullerAutoWidth : FBC.0x000001DD.0x00000001.NUTEK_DELTA_EDS_V101 v1.0 (OrderNumber=NUTEK_DELTA_V101)  [CAN1 -> Traverser.CAN2]
PullerPusher : FBC.0x000001DD.0x00000001.NUTEK_DELTA_EDS_V101 v1.0 (OrderNumber=NUTEK_DELTA_V101)  [CAN1 -> PullerAutoWidth.CAN2]
Traverser : FBC.0x000001DD.0x00000001.NUTEK_DELTA_EDS_V101 v1.0 (OrderNumber=NUTEK_DELTA_V101)  [CAN1 -> Lifter.CAN2]
X20BB57 : X20BB57 v1.1.1.0
  Connector IF1:
    Baudrate = 9600
    Parity = N
  Connector IF7:
    Baudrate = 1000000
    ActivateCanOpen = 1
    p100c_parametervalue = 1000
    p100d_parametervalue = 3
X20BM01 : X20BM01 v2.1.0.0  [X2X1 -> X20BM11d.X2X2]
X20BM11 : X20BM11 v1.0.0.1  [X2X1 -> X20BB57.IF6]
X20BM11a : X20BM11 v1.0.0.1  [X2X1 -> X20BM11.X2X2]
X20BM11b : X20BM11 v1.0.0.1  [X2X1 -> X20BM11a.X2X2]
X20BM11d : X20BM11 v1.0.0.1  [X2X1 -> X20BM11i.X2X2]
X20BM11e : X20BM11 v1.0.0.1  [X2X1 -> X20BM11f.X2X2]
X20BM11f : X20BM11 v1.0.0.1  [X2X1 -> X20BM01.X2X2]
X20BM11i : X20BM11 v1.0.0.1  [X2X1 -> X20BM11b.X2X2]
X20CP0483 : X20CP0483 v1.2.1.0  [SL -> X20BB57.SL1]
  Connector IF2:
    ActivateDevice = 1
    Mode = Manual
    InternetAddress = 192.168.0.2
    SubnetMask = 255.255.255.0
    Vnc1
    VncVcObjectName1 = Visu
    VncKeyMappingFile1 = VC\PS2-Keyboard.dis
    VncMaxConnections1 = 3
    VncRefreshRate1 = 100
    ActivateSnmp = 2
  ConfigurationID = NAELD004  // Unique Configuration ID. Required format: SpaCes at the beginning or end of the string are not permitted.
  UserPartitionSize = 150
  VolatileGlobalPvSize = 80000
  EnableUsbRemoteInstall = 1
  TimerDeviceType = SWIOTIMER
  Cyclic1Duration = 10000
  Cyclic1Tolerance = 10000
  Cyclic2Duration = 20000
  Cyclic2Tolerance = 20000
  Cyclic3Duration = 50000
  Cyclic3Tolerance = 50000
  Cyclic4Duration = 10000
  Cyclic4Tolerance = 10000
  Cyclic5Duration = 200000
  Cyclic5Tolerance = 200000
  Cyclic6Duration = 500000
  Cyclic6Tolerance = 500000
  Cyclic7Duration = 1000000
  Cyclic7Tolerance = 1000000
  Cyclic8Duration = 10000
  Cyclic8Tolerance = 10000
  FileDevice1
  FileDeviceName1 = F
  FileDevicePath1 = F:
  FileDevice2
  FileDeviceName2 = User
  FileDevicePath2 = F:\User
  FileDevice3
  FileDeviceName3 = Private
  FileDevicePath3 = F:\Private
  FileDevice4
  FileDeviceName4 = CustomerUser
  FileDevicePath4 = F:\User\UserMgmt
  FileDevice5
  FileDeviceName5 = ProdRcp
  FileDevicePath5 = F:\User\ProductRecipe
  FileDevice6
  FileDeviceName6 = MagRcp
  FileDevicePath6 = F:\User\MagazineRecipe
  FileDevice7
  FileDeviceName7 = Alarm
  FileDevicePath7 = F:\User\Alarm
  FileDevice8
  FileDeviceName8 = McParam
  FileDevicePath8 = F:\User\MachineParameter
  FileDevice9
  FileDeviceName9 = NtParam
  FileDevicePath9 = F:\Private\NutekParameter
  FileDevice10
  FileDeviceName10 = LibVer
  FileDevicePath10 = F:\User\LibrariesVersion
  FileDevice11
  FileDeviceName11 = Retain
  FileDevicePath11 = F:\User\Retain
  FileDevice12
  FileDeviceName12 = Log
  FileDevicePath12 = F:\User\Log
  FileDevice13
  FileDeviceName13 = LCS
  FileDevicePath13 = F:\User\LCS
  FileDevice14
  FileDeviceName14 = MpProdRcp
  FileDevicePath14 = F:\User\ProductRecipeXml
  FileDevice15
  FileDeviceName15 = MpNtParam
  FileDevicePath15 = F:\Private\NutekParameterXml
  FileDevice16
  FileDeviceName16 = MagRcp1
  FileDevicePath16 = F:\User\MagazineRecipe1
  FileDevice17
  FileDeviceName17 = Serial
  FileDevicePath17 = F:\User\Serial
  FileDevice18
  FileDeviceName18 = USB
  FileDevicePath18 = F:\User\Serial\USB
  FileDevice19
  FileDeviceName19 = RS232
  FileDevicePath19 = F:\User\Serial\RS232
  FtpUser1
  FtpUsername1 = NTAFTP
  FtpUserPassword1 = JmcONQZEIGyG0Pt+VekJRbxmc4fxS8REPwlCJguEtEY=  // NTA4BH
  FtpUserSalt1 = smKszLJT
  FTPAccessRight1 = 0
  FTPdevice1 = ALL
  FtpUser2
  FtpUsername2 = admin
  FtpUserPassword2 = GulCMI/jV0v16Ew6MS+jrzqmTLk+NRkNo3Y+jAhzSzY=  // admin
  FtpUserSalt2 = robUzvv7
  FTPAccessRight2 = 0
  FTPMSpath2 = User
  FtpUser3
  FtpUsername3 = LCS
  FtpUserPassword3 = 6XI8rzr3QlcLzq1fKGxRBMxxRW19t00F0QlEDJIXmLc=  // LCS
  FtpUserSalt3 = Xz6TWjSu
  FTPMSpath3 = User\LCS
  FtpUser4
  FtpUsername4 = user
  FtpUserPassword4 = WaRT3CuWXqstpfRIiz8AHLWR/dIjkiQ2KdDM3lRZC/M=  // user
  FtpUserSalt4 = iqIficTD
  FTPMSpath4 = User\ProductRecipeXml
  ActivateOpcUa = 1
  OpcUa_ConversationSecurityPolicy_EnableBasic256Rsa256 = 0
  OpcUaInformationModels_PV_Version = 1
X20DI9372_X2 : X20DI9372 v1.1.0.0  [SS1 -> X20TB12a.SS; SL -> X20BM11.SL1]
X20DI9372_X3 : X20DI9372 v1.1.0.0  [SS1 -> X20TB12b.SS; SL -> X20BM11a.SL1]
X20DI9372_X4 : X20DI9372 v1.1.0.0  [SS1 -> X20TB12c.SS; SL -> X20BM11b.SL1]
X20DI9372_X5 : X20DI9372 v1.1.0.0  [SS1 -> X20TB12k.SS; SL -> X20BM11i.SL1]
X20DO6321_X9 : X20DO6321 v1.1.0.0  [SS1 -> X20TB12e.SS; SL -> X20BM11d.SL1]
X20DO9321_X11 : X20DO9321 v1.1.0.0  [SS1 -> X20TB12h.SS; SL -> X20BM11f.SL1]
X20DO9321_X12 : X20DO9321 v1.1.0.0  [SS1 -> X20TB12g.SS; SL -> X20BM11e.SL1]
X20PS2100_X10 : X20PS2100 v1.2.0.0  [SS1 -> X20TB12f.SS; SL -> X20BM01.SL1]
X20PS9602_X1 : X20PS9602 v1.0.2.0  [PS -> X20BB57.PS1; SS1 -> X20TB12.SS]
X20TB12 : X20TB12 v1.0.0.0
X20TB12a : X20TB12 v1.0.0.0
X20TB12b : X20TB12 v1.0.0.0
X20TB12c : X20TB12 v1.0.0.0
X20TB12e : X20TB12 v1.0.0.0
X20TB12f : X20TB12 v1.0.0.0
X20TB12g : X20TB12 v1.0.0.0
X20TB12h : X20TB12 v1.0.0.0
X20TB12k : X20TB12 v1.0.0.0
```

### IoMap.iom - X20CP0483/IoMap.iom
```iecst
VAR_CONFIG
	::DInput:a_bPhysicalDI[1] AT %IX."X20DI9372_X2".DigitalInput01;
	::DInput:a_bPhysicalDI[2] AT %IX."X20DI9372_X2".DigitalInput02;
	::DInput:a_bPhysicalDI[3] AT %IX."X20DI9372_X2".DigitalInput03;
	::DInput:a_bPhysicalDI[4] AT %IX."X20DI9372_X2".DigitalInput04;
	::DInput:a_bPhysicalDI[5] AT %IX."X20DI9372_X2".DigitalInput05;
	::DInput:a_bPhysicalDI[6] AT %IX."X20DI9372_X2".DigitalInput06;
	::DInput:a_bPhysicalDI[7] AT %IX."X20DI9372_X2".DigitalInput07;
	::DInput:a_bPhysicalDI[8] AT %IX."X20DI9372_X2".DigitalInput08;
	::DInput:a_bPhysicalDI[9] AT %IX."X20DI9372_X2".DigitalInput09;
	::DInput:a_bPhysicalDI[10] AT %IX."X20DI9372_X2".DigitalInput10;
	::DInput:a_bPhysicalDI[11] AT %IX."X20DI9372_X2".DigitalInput11;
	::DInput:a_bPhysicalDI[12] AT %IX."X20DI9372_X2".DigitalInput12;
	::DInput:a_bPhysicalDI[13] AT %IX."X20DI9372_X3".DigitalInput01;
	::DInput:a_bPhysicalDI[14] AT %IX."X20DI9372_X3".DigitalInput02;
	::DInput:a_bPhysicalDI[15] AT %IX."X20DI9372_X3".DigitalInput03;
	::DInput:a_bPhysicalDI[16] AT %IX."X20DI9372_X3".DigitalInput04;
	::DInput:a_bPhysicalDI[17] AT %IX."X20DI9372_X3".DigitalInput05;
	::DInput:a_bPhysicalDI[18] AT %IX."X20DI9372_X3".DigitalInput06;
	::DInput:a_bPhysicalDI[19] AT %IX."X20DI9372_X3".DigitalInput07;
	::DInput:a_bPhysicalDI[20] AT %IX."X20DI9372_X3".DigitalInput08;
	::DInput:a_bPhysicalDI[21] AT %IX."X20DI9372_X3".DigitalInput09;
	::DInput:a_bPhysicalDI[22] AT %IX."X20DI9372_X3".DigitalInput10;
	::DInput:a_bPhysicalDI[23] AT %IX."X20DI9372_X3".DigitalInput11;
	::DInput:a_bPhysicalDI[24] AT %IX."X20DI9372_X3".DigitalInput12;
	::DInput:a_bPhysicalDI[25] AT %IX."X20DI9372_X4".DigitalInput01;
	::DInput:a_bPhysicalDI[26] AT %IX."X20DI9372_X4".DigitalInput02;
	::DInput:a_bPhysicalDI[27] AT %IX."X20DI9372_X4".DigitalInput03;
	::DInput:a_bPhysicalDI[28] AT %IX."X20DI9372_X4".DigitalInput04;
	::DInput:a_bPhysicalDI[29] AT %IX."X20DI9372_X4".DigitalInput05;
	::DInput:a_bPhysicalDI[30] AT %IX."X20DI9372_X4".DigitalInput06;
	::DInput:a_bPhysicalDI[31] AT %IX."X20DI9372_X4".DigitalInput07;
	::DInput:a_bPhysicalDI[32] AT %IX."X20DI9372_X4".DigitalInput08;
	::DInput:a_bPhysicalDI[33] AT %IX."X20DI9372_X4".DigitalInput09;
	::DInput:a_bPhysicalDI[34] AT %IX."X20DI9372_X4".DigitalInput10;
	::DInput:a_bPhysicalDI[35] AT %IX."X20DI9372_X4".DigitalInput11;
	::DInput:a_bPhysicalDI[36] AT %IX."X20DI9372_X4".DigitalInput12;
	::DOutput:a_bPhysicalDO[7] AT %QX."X20DO9321_X11".DigitalOutput01;
	::DOutput:a_bPhysicalDO[8] AT %QX."X20DO9321_X11".DigitalOutput02;
	::DOutput:a_bPhysicalDO[9] AT %QX."X20DO9321_X11".DigitalOutput03;
	::DOutput:a_bPhysicalDO[10] AT %QX."X20DO9321_X11".DigitalOutput04;
	::DOutput:a_bPhysicalDO[11] AT %QX."X20DO9321_X11".DigitalOutput05;
	::DOutput:a_bPhysicalDO[12] AT %QX."X20DO9321_X11".DigitalOutput06;
	::AWOpen:bModuleOK AT %IX."AutoWidth".ModuleOk;
	::AWOpen:tyParamInDriver.uiErrCode_603F AT %IW."AutoWidth".ErrorCode_603F;
	::AWOpen:tyParamOutDriver.uiCtrlword_6040 AT %QW."AutoWidth".Controlword_6040;
	::AWOpen:tyParamInDriver.uiStatword_6041 AT %IW."AutoWidth".Statusword_6041;
	::AWOpen:tyParamOutDriver.siModOfOpt_6060 AT %QB."AutoWidth".ModesOfOperation_6060;
	::AWOpen:tyParamInDriver.siModOfOptDisp_6061 AT %IB."AutoWidth".ModesOfOperationDisplay_6061;
	::AWOpen:tyParamInDriver.diActualPos_6064 AT %ID."AutoWidth".PositionActualValue_6064;
	::AWOpen:tyParamOutDriver.diTargetPos_607A AT %QD."AutoWidth".TargetPosition_607A;
	::AWOpen:tyParamOutDriver.udiMoveSpd_6081 AT %QD."AutoWidth".ProfileVelocity_6081;
	::AWOpen:tyParamOutDriver.siHmMethod_6098 AT %QB."AutoWidth".HomingMethod_6098;
	::AWOpen:tyParamInDriver.udiDigitalInputs_60FD AT %ID."AutoWidth".DigitalInputs_60FD;
	::AWOpen:tyParamOutDriver.diJogVel_60FF AT %QD."AutoWidth".TargetVelocity_60FF;
	::LifterBtm:bModuleOK AT %IX."Lifter".ModuleOk;
	::LifterBtm:tyParamInDriver.uiErrCode_603F AT %IW."Lifter".ErrorCode_603F;
	::LifterBtm:tyParamOutDriver.uiCtrlword_6040 AT %QW."Lifter".Controlword_6040;
	::LifterBtm:tyParamInDriver.uiStatword_6041 AT %IW."Lifter".Statusword_6041;
	::LifterBtm:tyParamOutDriver.siModOfOpt_6060 AT %QB."Lifter".ModesOfOperation_6060;
	::LifterBtm:tyParamInDriver.siModOfOptDisp_6061 AT %IB."Lifter".ModesOfOperationDisplay_6061;
	::LifterBtm:tyParamInDriver.diActualPos_6064 AT %ID."Lifter".PositionActualValue_6064;
	::LifterBtm:tyParamOutDriver.diTargetPos_607A AT %QD."Lifter".TargetPosition_607A;
	::LifterBtm:tyParamOutDriver.udiMoveSpd_6081 AT %QD."Lifter".ProfileVelocity_6081;
	::LifterBtm:tyParamOutDriver.siHmMethod_6098 AT %QB."Lifter".HomingMethod_6098;
	::LifterBtm:tyParamInDriver.udiDigitalInputs_60FD AT %ID."Lifter".DigitalInputs_60FD;
	::LifterBtm:tyParamOutDriver.diJogVel_60FF AT %QD."Lifter".TargetVelocity_60FF;
	::Trav:bModuleOK AT %IX."Traverser".ModuleOk;
	::Trav:tyParamInDriver.uiErrCode_603F AT %IW."Traverser".ErrorCode_603F;
	::Trav:tyParamOutDriver.uiCtrlword_6040 AT %QW."Traverser".Controlword_6040;
	::Trav:tyParamInDriver.uiStatword_6041 AT %IW."Traverser".Statusword_6041;
	::Trav:tyParamOutDriver.siModOfOpt_6060 AT %QB."Traverser".ModesOfOperation_6060;
	::Trav:tyParamInDriver.siModOfOptDisp_6061 AT %IB."Traverser".ModesOfOperationDisplay_6061;
	::Trav:tyParamInDriver.diActualPos_6064 AT %ID."Traverser".PositionActualValue_6064;
	::Trav:tyParamOutDriver.diTargetPos_607A AT %QD."Traverser".TargetPosition_607A;
	::Trav:tyParamOutDriver.udiMoveSpd_6081 AT %QD."Traverser".ProfileVelocity_6081;
	::Trav:tyParamOutDriver.siHmMethod_6098 AT %QB."Traverser".HomingMethod_6098;
	::Trav:tyParamInDriver.udiDigitalInputs_60FD AT %ID."Traverser".DigitalInputs_60FD;
	::Trav:tyParamOutDriver.diJogVel_60FF AT %QD."Traverser".TargetVelocity_60FF;
	::DOutput:a_bPhysicalDO[13] AT %QX."X20DO9321_X11".DigitalOutput07;
	::DOutput:a_bPhysicalDO[14] AT %QX."X20DO9321_X11".DigitalOutput08;
	::DOutput:a_bPhysicalDO[15] AT %QX."X20DO9321_X11".DigitalOutput09;
	::DOutput:a_bPhysicalDO[16] AT %QX."X20DO9321_X11".DigitalOutput10;
	::DOutput:a_bPhysicalDO[17] AT %QX."X20DO9321_X11".DigitalOutput11;
	::DOutput:a_bPhysicalDO[18] AT %QX."X20DO9321_X11".DigitalOutput12;
	::AWOpen:tyParamInDriver.uiErrCode_603F AT %IW."AutoWidth".Error_code_603F;
	::AWOpen:tyParamInDriver.siModOfOptDisp_6061 AT %IB."AutoWidth".Modes_of_operation_display_6061;
	::AWOpen:tyParamInDriver.diActualPos_6064 AT %ID."AutoWidth".Position_actual_value_6064;
	::AWOpen:tyParamInDriver.udiDigitalInputs_60FD AT %ID."AutoWidth".Digital_intputs_60FD;
	::AWOpen:tyParamOutDriver.siModOfOpt_6060 AT %QB."AutoWidth".Modes_of_operation_6060;
	::AWOpen:tyParamOutDriver.diTargetPos_607A AT %QD."AutoWidth".Target_position_607A;
	::AWOpen:tyParamOutDriver.udiMoveSpd_6081 AT %QD."AutoWidth".Profile_velocity_6081;
	::AWOpen:tyParamOutDriver.siHmMethod_6098 AT %QB."AutoWidth".Homing_method_6098;
	::AWOpen:tyParamOutDriver.diJogVel_60FF AT %QD."AutoWidth".Target_velocity_60FF;
	::LifterBtm:tyParamOutDriver.siModOfOpt_6060 AT %QB."Lifter".Modes_of_operation_6060;
	::LifterBtm:tyParamOutDriver.diTargetPos_607A AT %QD."Lifter".Target_position_607A;
	::LifterBtm:tyParamOutDriver.udiMoveSpd_6081 AT %QD."Lifter".Profile_velocity_6081;
	::LifterBtm:tyParamOutDriver.siHmMethod_6098 AT %QB."Lifter".Homing_method_6098;
	::LifterBtm:tyParamOutDriver.diJogVel_60FF AT %QD."Lifter".Target_velocity_60FF;
	::LifterBtm:tyParamInDriver.uiErrCode_603F AT %IW."Lifter".Error_code_603F;
	::LifterBtm:tyParamInDriver.siModOfOptDisp_6061 AT %IB."Lifter".Modes_of_operation_display_6061;
	::LifterBtm:tyParamInDriver.diActualPos_6064 AT %ID."Lifter".Position_actual_value_6064;
	::LifterBtm:tyParamInDriver.udiDigitalInputs_60FD AT %ID."Lifter".Digital_intputs_60FD;
	::Trav:tyParamOutDriver.siModOfOpt_6060 AT %QB."Traverser".Modes_of_operation_6060;
	::Trav:tyParamOutDriver.diTargetPos_607A AT %QD."Traverser".Target_position_607A;
	::Trav:tyParamOutDriver.udiMoveSpd_6081 AT %QD."Traverser".Profile_velocity_6081;
	::Trav:tyParamOutDriver.siHmMethod_6098 AT %QB."Traverser".Homing_method_6098;
	::Trav:tyParamOutDriver.diJogVel_60FF AT %QD."Traverser".Target_velocity_60FF;
	::Trav:tyParamInDriver.uiErrCode_603F AT %IW."Traverser".Error_code_603F;
	::Trav:tyParamInDriver.siModOfOptDisp_6061 AT %IB."Traverser".Modes_of_operation_display_6061;
	::Trav:tyParamInDriver.diActualPos_6064 AT %ID."Traverser".Position_actual_value_6064;
	::Trav:tyParamInDriver.udiDigitalInputs_60FD AT %ID."Traverser".Digital_intputs_60FD;
	::AWPushOrPu:bModuleOK AT %IX."PullerAutoWidth".ModuleOk;
	::AWPushOrPu:tyParamInDriver.uiErrCode_603F AT %IW."PullerAutoWidth".Error_code_603F;
	::AWPushOrPu:tyParamOutDriver.uiCtrlword_6040 AT %QW."PullerAutoWidth".Controlword_6040;
	::AWPushOrPu:tyParamInDriver.uiStatword_6041 AT %IW."PullerAutoWidth".Statusword_6041;
	::AWPushOrPu:tyParamInDriver.siModOfOptDisp_6061 AT %IB."PullerAutoWidth".Modes_of_operation_display_6061;
	::AWPushOrPu:tyParamInDriver.diActualPos_6064 AT %ID."PullerAutoWidth".Position_actual_value_6064;
	::AWPushOrPu:tyParamInDriver.udiDigitalInputs_60FD AT %ID."PullerAutoWidth".Digital_intputs_60FD;
	::AWPushOrPu:tyParamOutDriver.siModOfOpt_6060 AT %QB."PullerAutoWidth".Modes_of_operation_6060;
	::AWPushOrPu:tyParamOutDriver.diTargetPos_607A AT %QD."PullerAutoWidth".Target_position_607A;
	::AWPushOrPu:tyParamOutDriver.udiMoveSpd_6081 AT %QD."PullerAutoWidth".Profile_velocity_6081;
	::AWPushOrPu:tyParamOutDriver.siHmMethod_6098 AT %QB."PullerAutoWidth".Homing_method_6098;
	::AWPushOrPu:tyParamOutDriver.diJogVel_60FF AT %QD."PullerAutoWidth".Target_velocity_60FF;
	::DInput:a_bPhysicalDI[37] AT %IX."X20DI9372_X5".DigitalInput01;
	::DInput:a_bPhysicalDI[38] AT %IX."X20DI9372_X5".DigitalInput02;
	::DInput:a_bPhysicalDI[39] AT %IX."X20DI9372_X5".DigitalInput03;
	::DInput:a_bPhysicalDI[40] AT %IX."X20DI9372_X5".DigitalInput04;
	::DInput:a_bPhysicalDI[41] AT %IX."X20DI9372_X5".DigitalInput05;
	::DInput:a_bPhysicalDI[42] AT %IX."X20DI9372_X5".DigitalInput06;
	::DInput:a_bPhysicalDI[43] AT %IX."X20DI9372_X5".DigitalInput07;
	::DInput:a_bPhysicalDI[44] AT %IX."X20DI9372_X5".DigitalInput08;
	::DInput:a_bPhysicalDI[45] AT %IX."X20DI9372_X5".DigitalInput09;
	::DInput:a_bPhysicalDI[46] AT %IX."X20DI9372_X5".DigitalInput10;
	::DInput:a_bPhysicalDI[47] AT %IX."X20DI9372_X5".DigitalInput11;
	::DInput:a_bPhysicalDI[48] AT %IX."X20DI9372_X5".DigitalInput12;
	::DOutput:a_bPhysicalDO[1] AT %QX."X20DO6321_X11".DigitalOutput01;
	::DOutput:a_bPhysicalDO[2] AT %QX."X20DO6321_X11".DigitalOutput02;
	::DOutput:a_bPhysicalDO[3] AT %QX."X20DO6321_X11".DigitalOutput03;
	::DOutput:a_bPhysicalDO[4] AT %QX."X20DO6321_X11".DigitalOutput04;
	::DOutput:a_bPhysicalDO[5] AT %QX."X20DO6321_X11".DigitalOutput05;
	::DOutput:a_bPhysicalDO[6] AT %QX."X20DO6321_X11".DigitalOutput06;
	::DOutput:a_bPhysicalDO[19] AT %QX."X20DO9321_X12".DigitalOutput01;
	::DOutput:a_bPhysicalDO[20] AT %QX."X20DO9321_X12".DigitalOutput02;
	::DOutput:a_bPhysicalDO[21] AT %QX."X20DO9321_X12".DigitalOutput03;
	::DOutput:a_bPhysicalDO[22] AT %QX."X20DO9321_X12".DigitalOutput04;
	::DOutput:a_bPhysicalDO[23] AT %QX."X20DO9321_X12".DigitalOutput05;
	::DOutput:a_bPhysicalDO[24] AT %QX."X20DO9321_X12".DigitalOutput06;
	::DOutput:a_bPhysicalDO[25] AT %QX."X20DO9321_X12".DigitalOutput07;
	::DOutput:a_bPhysicalDO[26] AT %QX."X20DO9321_X12".DigitalOutput08;
	::DOutput:a_bPhysicalDO[27] AT %QX."X20DO9321_X12".DigitalOutput09;
	::DOutput:a_bPhysicalDO[28] AT %QX."X20DO9321_X12".DigitalOutput10;
	::DOutput:a_bPhysicalDO[29] AT %QX."X20DO9321_X12".DigitalOutput11;
	::DOutput:a_bPhysicalDO[30] AT %QX."X20DO9321_X12".DigitalOutput12;
	::DOutput:a_bPhysicalDO[1] AT %QX."X20DO6321_X9".DigitalOutput01;
	::DOutput:a_bPhysicalDO[2] AT %QX."X20DO6321_X9".DigitalOutput02;
	::DOutput:a_bPhysicalDO[3] AT %QX."X20DO6321_X9".DigitalOutput03;
	::DOutput:a_bPhysicalDO[4] AT %QX."X20DO6321_X9".DigitalOutput04;
	::DOutput:a_bPhysicalDO[5] AT %QX."X20DO6321_X9".DigitalOutput05;
	::DOutput:a_bPhysicalDO[6] AT %QX."X20DO6321_X9".DigitalOutput06;
	::AWPushOrPu:tyParamInDriver.siModOfOptDisp_6061 AT %IB."PullerAutoWidth".ModesOfOperationDisplay_6061;
	::AWPushOrPu:tyParamInDriver.diActualPos_6064 AT %ID."PullerAutoWidth".PositionActualValue_6064;
	::AWPushOrPu:tyParamInDriver.udiDigitalInputs_60FD AT %ID."PullerAutoWidth".DigitalInputs_60FD;
	::AWPushOrPu:tyParamOutDriver.siModOfOpt_6060 AT %QB."PullerAutoWidth".ModesOfOperation_6060;
	::AWPushOrPu:tyParamOutDriver.diTargetPos_607A AT %QD."PullerAutoWidth".TargetPosition_607A;
	::AWPushOrPu:tyParamOutDriver.udiMoveSpd_6081 AT %QD."PullerAutoWidth".ProfileVelocity_6081;
	::AWPushOrPu:tyParamOutDriver.siHmMethod_6098 AT %QB."PullerAutoWidth".HomingMethod_6098;
	::AWPushOrPu:tyParamOutDriver.diJogVel_60FF AT %QD."PullerAutoWidth".TargetVelocity_60FF;
	::PullerPush:bModuleOK AT %IX."PullerPusher".ModuleOk;
	::PullerPush:tyParamInDriver.uiErrCode_603F AT %IW."PullerPusher".ErrorCode_603F;
	::PullerPush:tyParamInDriver.uiStatword_6041 AT %IW."PullerPusher".Statusword_6041;
	::PullerPush:tyParamInDriver.siModOfOptDisp_6061 AT %IB."PullerPusher".ModesOfOperationDisplay_6061;
	::PullerPush:tyParamInDriver.udiDigitalInputs_60FD AT %ID."PullerPusher".DigitalInputs_60FD;
	::PullerPush:tyParamOutDriver.uiCtrlword_6040 AT %QW."PullerPusher".Controlword_6040;
	::PullerPush:tyParamOutDriver.siModOfOpt_6060 AT %QB."PullerPusher".ModesOfOperation_6060;
	::PullerPush:tyParamInDriver.diActualPos_6064 AT %ID."PullerPusher".PositionActualValue_6064;
	::PullerPush:tyParamOutDriver.diTargetPos_607A AT %QD."PullerPusher".TargetPosition_607A;
	::PullerPush:tyParamOutDriver.udiMoveSpd_6081 AT %QD."PullerPusher".ProfileVelocity_6081;
	::PullerPush:tyParamOutDriver.siHmMethod_6098 AT %QB."PullerPusher".HomingMethod_6098;
	::PullerPush:tyParamOutDriver.diJogVel_60FF AT %QD."PullerPusher".TargetVelocity_60FF;
	::AWPushOrPu:tyParamInDriver.uiErrCode_603F AT %IW."PullerAutoWidth".ErrorCode_603F;
END_VAR
```

## Configuration 3Mag_RotMtrPuller_Delta

### Task classes (Cpu.sw)
```
Cyclic#1 (cycle 10000 us, tolerance 10000 us):
  DInput <- DInput.DInput.prg
  DOutput <- DOutput.DOutput.prg
Cyclic#2 (cycle 20000 us, tolerance 20000 us):
  BarcodeRdr <- USBBarcodeRdr.BarcodeRdr.prg
  PullConv <- Conv.PullConv.prg
  MagConv2Cl <- MagConv.MagConv2Clp1.prg
  MagConv2C1 <- MagConv.MagConv2Clp2.prg
  MagConv2C2 <- MagConv.MagConv2Clp3.prg
  MagConv2C3 <- MagConv.MagConv2Clp4.prg
  MtrPshr <- MtrPshr.MtrPshr.prg
  PullerPush <- CANOpenServo.PullerPusher.PullerPusher.prg
Cyclic#3 (cycle 50000 us, tolerance 50000 us):
  UI <- UI.UI.prg
  Startup <- Startup.Startup.prg
  General <- General.General.prg
  UsrFolder <- UsrFolder.UsrFolder.prg
  LibVer <- LibVer.LibVer.prg
  Time <- Time.Time.prg
  HWInfo <- HWInfo.HWInfo.prg
  TLBuz <- TLBuz.TLBuz.prg
  Alarm <- Alarm.Alarm.prg
  RstErr <- RstErr.RstErr.prg
  ProdRcp <- ProdRcp.ProdRcp.prg
  MpProdRcp <- MpProdRcp.MpProdRcp.prg
  MagRcp <- MagRcp.MagRcp.prg
  MagRcp1 <- MagRcp.MagRcp1.prg
  McParam <- McParam.McParam.prg
  NtParam <- NtParam.NtParam.prg
  UsrMgmt <- UsrMgmt.UsrMgmt.prg
  Buffer1 <- Buffer.Buffer1.prg
  Buffer2 <- Buffer.Buffer2.prg
  Buffer3 <- Buffer.Buffer3.prg
  Buffer4 <- Buffer.Buffer4.prg
  USSMEMA1 <- SMEMA.USSMEMA1.prg
  USSMEMA2 <- SMEMA.USSMEMA2.prg
  USSMEMA3 <- SMEMA.USSMEMA3.prg
  USSMEMA4 <- SMEMA.USSMEMA4.prg
  DSSMEMA1 <- SMEMA.DSSMEMA1.prg
  DSSMEMA2 <- SMEMA.DSSMEMA2.prg
  DSSMEMA3 <- SMEMA.DSSMEMA3.prg
  DSSMEMA4 <- SMEMA.DSSMEMA4.prg
  DSSMEMAA <- SMEMA.DSSMEMAA.prg
  DSSMEMAB <- SMEMA.DSSMEMAB.prg
  Pneu2SenIn <- Pneu.Pneu2SenInShutter.prg
  Pneu2SenOu <- Pneu.Pneu2SenOutShutter.prg
  Pneu2SenO1 <- Pneu.Pneu2SenOutShutter2.prg
  Pneu2SenPu <- Pneu.Pneu2SenPuller.prg
  Pneu2SenI1 <- Pneu.Pneu2SenInShutter2.prg
  Pneu2SenI2 <- Pneu.Pneu2SenInShutter3.prg
  Pneu2SenMa <- Pneu.MagSafetyBar.Pneu2SenMag1SafetyBar.prg
  Pneu2SenM1 <- Pneu.MagSafetyBar.Pneu2SenMag2SafetyBar.prg
  Pneu2SenM2 <- Pneu.MagSafetyBar.Pneu2SenMag3SafetyBar.prg
  Pneu2SenM3 <- Pneu.MagSafetyBar.Pneu2SenMag4SafetyBar.prg
  AWPushOrPu <- CANOpenServo.AW.AWPushOrPuller.prg
  AWOpen <- CANOpenServo.AW.AWOpen.prg
  Trav <- CANOpenServo.Trav.Trav.prg
  LifterBtm <- CANOpenServo.Lifter.LifterBtm.prg
  Hermes <- Hermes.Hermes.prg
  DSHermesA <- Hermes.DSHermesA.prg
  DSHermesB <- Hermes.DSHermesB.prg
  RmtHermes <- Hermes.RmtHermes.prg
  SvyHermes <- Hermes.SvyHermes.prg
  LFLeader <- LF.LFLeader.prg
  LFFollower <- LF.LFFollower.prg
  Follower1 <- LF.Follower1.prg
  Follower2 <- LF.Follower2.prg
  LCS <- LCS.LCS.prg
  LCSMngRcp <- LCS.LCSMngRcp.prg
  LCSLF <- LCS.LCSLF.prg
  Ops <- Operations.Ops.prg
  OpsTravLif <- Operations.OpsTravLifLD.prg
  OpsMagConv <- Operations.OpsMagConvLD1.prg
  OpsMagCon1 <- Operations.OpsMagConvLD2.prg
  OpsMagCon2 <- Operations.OpsMagConvLD3.prg
  OpsMagCon3 <- Operations.OpsMagConvLD4.prg
  OpsLifMagL <- Operations.OpsLifMagLD.prg
  AGV <- AGVCom.AGV.prg
  AGV1 <- AGVCom.AGV1.prg
  AGV2 <- AGVCom.AGV2.prg
  AGV3 <- AGVCom.AGV3.prg
  AGV4 <- AGVCom.AGV4.prg
  Pneu2SenSe <- Pneu.SelClamp.Pneu2SenSelClamp1.prg
  Pneu2SenS1 <- Pneu.SelClamp.Pneu2SenSelClamp2.prg
  Pneu2SenS2 <- Pneu.SelClamp.Pneu2SenSelClamp3.prg
  Pneu2SenS3 <- Pneu.SelClamp.Pneu2SenSelClamp4.prg
  Simu <- Simulation.Simu.prg
  USSOT1 <- SOT.USSOT1.prg
  DSSOT1 <- SOT.DSSOT1.prg
  USSOT2 <- SOT.USSOT2.prg
  DSSOT2 <- SOT.DSSOT2.prg
  USSOT3 <- SOT.USSOT3.prg
  DSSOT3 <- SOT.DSSOT3.prg
  USSOT4 <- SOT.USSOT4.prg
  DSSOT4 <- SOT.DSSOT4.prg
  Machine <- Machine.Machine.prg
  Machine1 <- Machine.Machine1.prg
  Frame <- RS232.DVFrame.Frame.prg
  AutoRcp <- AutoRcp.AutoRcp.prg
  PneuExtSen <- Pneu.Trolley.PneuExtSenTrolley.prg
  PneuExtSe1 <- Pneu.Trolley.PneuExtSenTrolley2.prg
DataObjects: Acp10sys
VcDataObjects: Visu <- UI.Visu.dob
Binaries: vccdt, vccbmp, Visu03, vcfile, arial, vctcal, arialxsr, vcmgr, visvc, vccstr, vcbclass, vccbtn, vcgclass, vcdsint, vcnet, vccline, vcshared, vccddbox, arialbd, vccnum, vcpdvnc, vcpdsw, vccslider, vccbar, vcctext, Visu01, arialbi, vcfntttf, vccovl, vccshape, vcalarm, Visu02, vcrt, udbdef, vccpopup, vcdsloc, vcchspot, TCData, vcpkat, vcpfgen, arsvcreg, vccalarm, User, sysconf, ashwac, ashwd, Role, asfw, arconfig, iomap, Config, vcpfar00, acp10cfg, Acp10map, OpcUaMap
Libraries: standard, runtime, NtLF, astime, asstring, operator, AsIecCon, AsCANopen, visapi, FileIO, AsIODiag, AsMem, dvframe, AsOpcUac, AsARCfg, sys_lib, AsTCP, MpRecipe, AsFltGen, brsystem, NtBuffer, NtConv, NtFileIO, NtLogFile, NtSMEMA, NtMem, NtMessage, NtOPCUA, NtOvenInfo, NtPneu, NtRS232, NtTLBuz, NtTCP, NtVersion, MpCom, MpBase, AsUSB, NtSOT, NtUSB, NtRecipe, NtGeneral, NtUI, NtMotion, sprintf, NtHermes, vcresman, dataobj, asmath, powerlnk
```

### Hardware
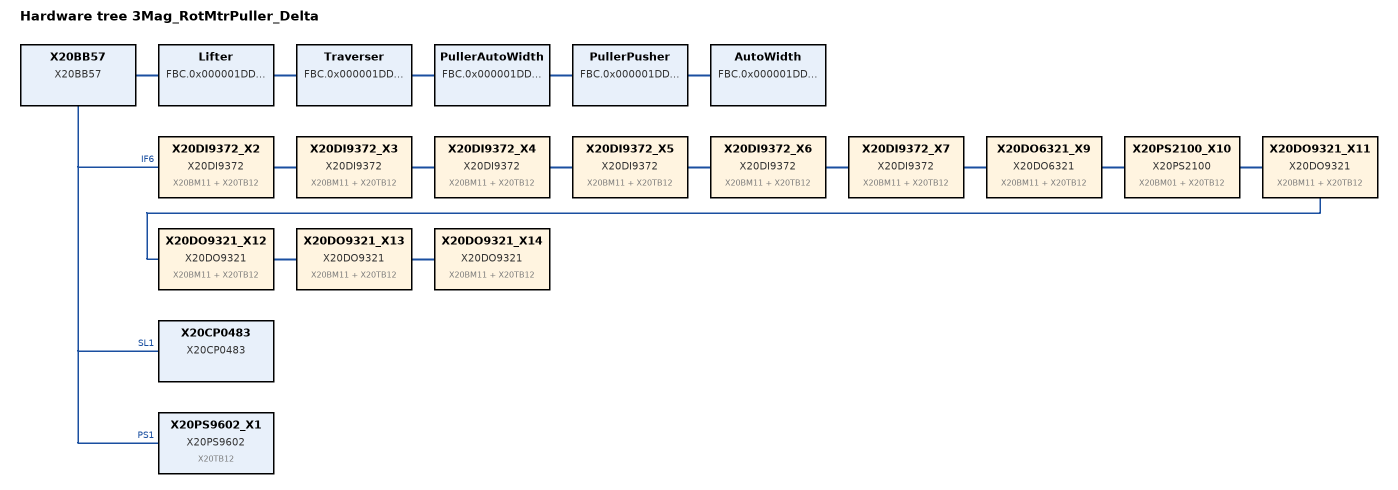
```
AutoWidth : FBC.0x000001DD.0x00000001.NUTEK_DELTA_EDS_V101 v1.0 (OrderNumber=NUTEK_DELTA_V101)  [CAN1 -> PullerPusher.CAN2 (NodeNumber=16)]
Lifter : FBC.0x000001DD.0x00000001.NUTEK_DELTA_EDS_V101 v1.0 (OrderNumber=NUTEK_DELTA_V101)  [CAN1 -> X20BB57.IF7 (NodeNumber=17)]
PullerAutoWidth : FBC.0x000001DD.0x00000001.NUTEK_DELTA_EDS_V101 v1.0 (OrderNumber=NUTEK_DELTA_V101)  [CAN1 -> Traverser.CAN2]
PullerPusher : FBC.0x000001DD.0x00000001.NUTEK_DELTA_EDS_V101 v1.0 (OrderNumber=NUTEK_DELTA_V101)  [CAN1 -> PullerAutoWidth.CAN2]
Traverser : FBC.0x000001DD.0x00000001.NUTEK_DELTA_EDS_V101 v1.0 (OrderNumber=NUTEK_DELTA_V101)  [CAN1 -> Lifter.CAN2]
X20BB57 : X20BB57 v1.1.1.0
  Connector IF1:
    Baudrate = 9600
    Parity = N
  Connector IF7:
    Baudrate = 1000000
    ActivateCanOpen = 1
    p100c_parametervalue = 1000
    p100d_parametervalue = 3
X20BM01 : X20BM01 v2.1.0.0  [X2X1 -> X20BM11d.X2X2]
X20BM11 : X20BM11 v1.0.0.1  [X2X1 -> X20BB57.IF6]
X20BM11a : X20BM11 v1.0.0.1  [X2X1 -> X20BM11.X2X2]
X20BM11b : X20BM11 v1.0.0.1  [X2X1 -> X20BM11a.X2X2]
X20BM11c : X20BM11 v1.0.0.1  [X2X1 -> X20BM11e.X2X2]
X20BM11d : X20BM11 v1.0.0.1  [X2X1 -> X20BM11g.X2X2]
X20BM11e : X20BM11 v1.0.0.1  [X2X1 -> X20BM11f.X2X2]
X20BM11f : X20BM11 v1.0.0.1  [X2X1 -> X20BM01.X2X2]
X20BM11g : X20BM11 v1.0.0.1  [X2X1 -> X20BM11j.X2X2]
X20BM11i : X20BM11 v1.0.0.1  [X2X1 -> X20BM11b.X2X2]
X20BM11j : X20BM11 v1.0.0.1  [X2X1 -> X20BM11i.X2X2]
X20BM11k : X20BM11 v1.0.0.1  [X2X1 -> X20BM11c.X2X2]
X20CP0483 : X20CP0483 v1.2.1.0  [SL -> X20BB57.SL1]
  Connector IF2:
    ActivateDevice = 1
    Mode = Manual
    InternetAddress = 192.168.0.32
    SubnetMask = 255.255.255.0
    InaNodeNumber = 32
    Vnc1
    VncVcObjectName1 = Visu
    VncKeyMappingFile1 = VC\PS2-Keyboard.dis
    VncMaxConnections1 = 3
    VncRefreshRate1 = 100
    ActivateSnmp = 2
  ConfigurationID = NAELD004  // Unique Configuration ID. Required format: SpaCes at the beginning or end of the string are not permitted.
  UserPartitionSize = 150
  VolatileGlobalPvSize = 80000
  EnableUsbRemoteInstall = 1
  TimerDeviceType = SWIOTIMER
  Cyclic1Duration = 10000
  Cyclic1Tolerance = 10000
  Cyclic2Duration = 20000
  Cyclic2Tolerance = 20000
  Cyclic3Duration = 50000
  Cyclic3Tolerance = 50000
  Cyclic4Duration = 10000
  Cyclic4Tolerance = 10000
  Cyclic5Duration = 200000
  Cyclic5Tolerance = 200000
  Cyclic6Duration = 500000
  Cyclic6Tolerance = 500000
  Cyclic7Duration = 1000000
  Cyclic7Tolerance = 1000000
  Cyclic8Duration = 10000
  Cyclic8Tolerance = 10000
  FileDevice1
  FileDeviceName1 = F
  FileDevicePath1 = F:
  FileDevice2
  FileDeviceName2 = User
  FileDevicePath2 = F:\User
  FileDevice3
  FileDeviceName3 = Private
  FileDevicePath3 = F:\Private
  FileDevice4
  FileDeviceName4 = CustomerUser
  FileDevicePath4 = F:\User\UserMgmt
  FileDevice5
  FileDeviceName5 = ProdRcp
  FileDevicePath5 = F:\User\ProductRecipe
  FileDevice6
  FileDeviceName6 = MagRcp
  FileDevicePath6 = F:\User\MagazineRecipe
  FileDevice7
  FileDeviceName7 = Alarm
  FileDevicePath7 = F:\User\Alarm
  FileDevice8
  FileDeviceName8 = McParam
  FileDevicePath8 = F:\User\MachineParameter
  FileDevice9
  FileDeviceName9 = NtParam
  FileDevicePath9 = F:\Private\NutekParameter
  FileDevice10
  FileDeviceName10 = LibVer
  FileDevicePath10 = F:\User\LibrariesVersion
  FileDevice11
  FileDeviceName11 = Retain
  FileDevicePath11 = F:\User\Retain
  FileDevice12
  FileDeviceName12 = Log
  FileDevicePath12 = F:\User\Log
  FileDevice13
  FileDeviceName13 = LCS
  FileDevicePath13 = F:\User\LCS
  FileDevice14
  FileDeviceName14 = MpProdRcp
  FileDevicePath14 = F:\User\ProductRecipeXml
  FileDevice15
  FileDeviceName15 = MpNtParam
  FileDevicePath15 = F:\Private\NutekParameterXml
  FileDevice16
  FileDeviceName16 = MagRcp1
  FileDevicePath16 = F:\User\MagazineRecipe1
  FileDevice17
  FileDeviceName17 = Serial
  FileDevicePath17 = F:\User\Serial
  FileDevice18
  FileDeviceName18 = USB
  FileDevicePath18 = F:\User\Serial\USB
  FileDevice19
  FileDeviceName19 = RS232
  FileDevicePath19 = F:\User\Serial\RS232
  FtpUser1
  FtpUsername1 = NTAFTP
  FtpUserPassword1 = JmcONQZEIGyG0Pt+VekJRbxmc4fxS8REPwlCJguEtEY=  // NTA4BH
  FtpUserSalt1 = smKszLJT
  FTPAccessRight1 = 0
  FTPdevice1 = ALL
  FtpUser2
  FtpUsername2 = admin
  FtpUserPassword2 = GulCMI/jV0v16Ew6MS+jrzqmTLk+NRkNo3Y+jAhzSzY=  // admin
  FtpUserSalt2 = robUzvv7
  FTPAccessRight2 = 0
  FTPMSpath2 = User
  FtpUser3
  FtpUsername3 = LCS
  FtpUserPassword3 = 6XI8rzr3QlcLzq1fKGxRBMxxRW19t00F0QlEDJIXmLc=  // LCS
  FtpUserSalt3 = Xz6TWjSu
  FTPMSpath3 = User\LCS
  FtpUser4
  FtpUsername4 = user
  FtpUserPassword4 = WaRT3CuWXqstpfRIiz8AHLWR/dIjkiQ2KdDM3lRZC/M=  // user
  FtpUserSalt4 = iqIficTD
  FTPMSpath4 = User\ProductRecipeXml
  ActivateOpcUa = 1
  OpcUa_ConversationSecurityPolicy_EnableBasic256Rsa256 = 0
  OpcUaInformationModels_PV_Version = 1
X20DI9372_X2 : X20DI9372 v1.1.0.0  [SS1 -> X20TB12a.SS; SL -> X20BM11.SL1]
X20DI9372_X3 : X20DI9372 v1.1.0.0  [SS1 -> X20TB12b.SS; SL -> X20BM11a.SL1]
X20DI9372_X4 : X20DI9372 v1.1.0.0  [SS1 -> X20TB12c.SS; SL -> X20BM11b.SL1]
X20DI9372_X5 : X20DI9372 v1.1.0.0  [SS1 -> X20TB12k.SS; SL -> X20BM11i.SL1]
X20DI9372_X6 : X20DI9372 v1.1.0.0  [SS1 -> X20TB12l.SS; SL -> X20BM11j.SL1]
X20DI9372_X7 : X20DI9372 v1.1.0.0  [SS1 -> X20TB12i.SS; SL -> X20BM11g.SL1]
X20DO6321_X9 : X20DO6321 v1.1.0.0  [SS1 -> X20TB12e.SS; SL -> X20BM11d.SL1]
X20DO9321_X11 : X20DO9321 v1.1.0.0  [SS1 -> X20TB12h.SS; SL -> X20BM11f.SL1]
X20DO9321_X12 : X20DO9321 v1.1.0.0  [SS1 -> X20TB12g.SS; SL -> X20BM11e.SL1]
X20DO9321_X13 : X20DO9321 v1.1.0.0  [SS1 -> X20TB12d.SS; SL -> X20BM11c.SL1]
X20DO9321_X14 : X20DO9321 v1.1.0.0  [SS1 -> X20TB12m.SS; SL -> X20BM11k.SL1]
X20PS2100_X10 : X20PS2100 v1.2.0.0  [SS1 -> X20TB12f.SS; SL -> X20BM01.SL1]
X20PS9602_X1 : X20PS9602 v1.0.2.0  [PS -> X20BB57.PS1; SS1 -> X20TB12.SS]
X20TB12 : X20TB12 v1.0.0.0
X20TB12a : X20TB12 v1.0.0.0
X20TB12b : X20TB12 v1.0.0.0
X20TB12c : X20TB12 v1.0.0.0
X20TB12d : X20TB12 v1.0.0.0
X20TB12e : X20TB12 v1.0.0.0
X20TB12f : X20TB12 v1.0.0.0
X20TB12g : X20TB12 v1.0.0.0
X20TB12h : X20TB12 v1.0.0.0
X20TB12i : X20TB12 v1.0.0.0
X20TB12k : X20TB12 v1.0.0.0
X20TB12l : X20TB12 v1.0.0.0
X20TB12m : X20TB12 v1.0.0.0
```

### IoMap.iom - X20CP0483/IoMap.iom
```iecst
VAR_CONFIG
	::DInput:a_bPhysicalDI[1] AT %IX."X20DI9372_X2".DigitalInput01;
	::DInput:a_bPhysicalDI[2] AT %IX."X20DI9372_X2".DigitalInput02;
	::DInput:a_bPhysicalDI[3] AT %IX."X20DI9372_X2".DigitalInput03;
	::DInput:a_bPhysicalDI[4] AT %IX."X20DI9372_X2".DigitalInput04;
	::DInput:a_bPhysicalDI[5] AT %IX."X20DI9372_X2".DigitalInput05;
	::DInput:a_bPhysicalDI[6] AT %IX."X20DI9372_X2".DigitalInput06;
	::DInput:a_bPhysicalDI[7] AT %IX."X20DI9372_X2".DigitalInput07;
	::DInput:a_bPhysicalDI[8] AT %IX."X20DI9372_X2".DigitalInput08;
	::DInput:a_bPhysicalDI[9] AT %IX."X20DI9372_X2".DigitalInput09;
	::DInput:a_bPhysicalDI[10] AT %IX."X20DI9372_X2".DigitalInput10;
	::DInput:a_bPhysicalDI[11] AT %IX."X20DI9372_X2".DigitalInput11;
	::DInput:a_bPhysicalDI[12] AT %IX."X20DI9372_X2".DigitalInput12;
	::DInput:a_bPhysicalDI[13] AT %IX."X20DI9372_X3".DigitalInput01;
	::DInput:a_bPhysicalDI[14] AT %IX."X20DI9372_X3".DigitalInput02;
	::DInput:a_bPhysicalDI[15] AT %IX."X20DI9372_X3".DigitalInput03;
	::DInput:a_bPhysicalDI[16] AT %IX."X20DI9372_X3".DigitalInput04;
	::DInput:a_bPhysicalDI[17] AT %IX."X20DI9372_X3".DigitalInput05;
	::DInput:a_bPhysicalDI[18] AT %IX."X20DI9372_X3".DigitalInput06;
	::DInput:a_bPhysicalDI[19] AT %IX."X20DI9372_X3".DigitalInput07;
	::DInput:a_bPhysicalDI[20] AT %IX."X20DI9372_X3".DigitalInput08;
	::DInput:a_bPhysicalDI[21] AT %IX."X20DI9372_X3".DigitalInput09;
	::DInput:a_bPhysicalDI[22] AT %IX."X20DI9372_X3".DigitalInput10;
	::DInput:a_bPhysicalDI[23] AT %IX."X20DI9372_X3".DigitalInput11;
	::DInput:a_bPhysicalDI[24] AT %IX."X20DI9372_X3".DigitalInput12;
	::DInput:a_bPhysicalDI[25] AT %IX."X20DI9372_X4".DigitalInput01;
	::DInput:a_bPhysicalDI[26] AT %IX."X20DI9372_X4".DigitalInput02;
	::DInput:a_bPhysicalDI[27] AT %IX."X20DI9372_X4".DigitalInput03;
	::DInput:a_bPhysicalDI[28] AT %IX."X20DI9372_X4".DigitalInput04;
	::DInput:a_bPhysicalDI[29] AT %IX."X20DI9372_X4".DigitalInput05;
	::DInput:a_bPhysicalDI[30] AT %IX."X20DI9372_X4".DigitalInput06;
	::DInput:a_bPhysicalDI[31] AT %IX."X20DI9372_X4".DigitalInput07;
	::DInput:a_bPhysicalDI[32] AT %IX."X20DI9372_X4".DigitalInput08;
	::DInput:a_bPhysicalDI[33] AT %IX."X20DI9372_X4".DigitalInput09;
	::DInput:a_bPhysicalDI[34] AT %IX."X20DI9372_X4".DigitalInput10;
	::DInput:a_bPhysicalDI[35] AT %IX."X20DI9372_X4".DigitalInput11;
	::DInput:a_bPhysicalDI[36] AT %IX."X20DI9372_X4".DigitalInput12;
	::DOutput:a_bPhysicalDO[7] AT %QX."X20DO9321_X11".DigitalOutput01;
	::DOutput:a_bPhysicalDO[8] AT %QX."X20DO9321_X11".DigitalOutput02;
	::DOutput:a_bPhysicalDO[9] AT %QX."X20DO9321_X11".DigitalOutput03;
	::DOutput:a_bPhysicalDO[10] AT %QX."X20DO9321_X11".DigitalOutput04;
	::DOutput:a_bPhysicalDO[11] AT %QX."X20DO9321_X11".DigitalOutput05;
	::DOutput:a_bPhysicalDO[12] AT %QX."X20DO9321_X11".DigitalOutput06;
	::AWOpen:bModuleOK AT %IX."AutoWidth".ModuleOk;
	::AWOpen:tyParamInDriver.uiErrCode_603F AT %IW."AutoWidth".ErrorCode_603F;
	::AWOpen:tyParamOutDriver.uiCtrlword_6040 AT %QW."AutoWidth".Controlword_6040;
	::AWOpen:tyParamInDriver.uiStatword_6041 AT %IW."AutoWidth".Statusword_6041;
	::AWOpen:tyParamOutDriver.siModOfOpt_6060 AT %QB."AutoWidth".ModesOfOperation_6060;
	::AWOpen:tyParamInDriver.siModOfOptDisp_6061 AT %IB."AutoWidth".ModesOfOperationDisplay_6061;
	::AWOpen:tyParamInDriver.diActualPos_6064 AT %ID."AutoWidth".PositionActualValue_6064;
	::AWOpen:tyParamOutDriver.diTargetPos_607A AT %QD."AutoWidth".TargetPosition_607A;
	::AWOpen:tyParamOutDriver.udiMoveSpd_6081 AT %QD."AutoWidth".ProfileVelocity_6081;
	::AWOpen:tyParamOutDriver.siHmMethod_6098 AT %QB."AutoWidth".HomingMethod_6098;
	::AWOpen:tyParamInDriver.udiDigitalInputs_60FD AT %ID."AutoWidth".DigitalInputs_60FD;
	::AWOpen:tyParamOutDriver.diJogVel_60FF AT %QD."AutoWidth".TargetVelocity_60FF;
	::LifterBtm:bModuleOK AT %IX."Lifter".ModuleOk;
	::LifterBtm:tyParamInDriver.uiErrCode_603F AT %IW."Lifter".ErrorCode_603F;
	::LifterBtm:tyParamOutDriver.uiCtrlword_6040 AT %QW."Lifter".Controlword_6040;
	::LifterBtm:tyParamInDriver.uiStatword_6041 AT %IW."Lifter".Statusword_6041;
	::LifterBtm:tyParamOutDriver.siModOfOpt_6060 AT %QB."Lifter".ModesOfOperation_6060;
	::LifterBtm:tyParamInDriver.siModOfOptDisp_6061 AT %IB."Lifter".ModesOfOperationDisplay_6061;
	::LifterBtm:tyParamInDriver.diActualPos_6064 AT %ID."Lifter".PositionActualValue_6064;
	::LifterBtm:tyParamOutDriver.diTargetPos_607A AT %QD."Lifter".TargetPosition_607A;
	::LifterBtm:tyParamOutDriver.udiMoveSpd_6081 AT %QD."Lifter".ProfileVelocity_6081;
	::LifterBtm:tyParamOutDriver.siHmMethod_6098 AT %QB."Lifter".HomingMethod_6098;
	::LifterBtm:tyParamInDriver.udiDigitalInputs_60FD AT %ID."Lifter".DigitalInputs_60FD;
	::LifterBtm:tyParamOutDriver.diJogVel_60FF AT %QD."Lifter".TargetVelocity_60FF;
	::Trav:bModuleOK AT %IX."Traverser".ModuleOk;
	::Trav:tyParamInDriver.uiErrCode_603F AT %IW."Traverser".ErrorCode_603F;
	::Trav:tyParamOutDriver.uiCtrlword_6040 AT %QW."Traverser".Controlword_6040;
	::Trav:tyParamInDriver.uiStatword_6041 AT %IW."Traverser".Statusword_6041;
	::Trav:tyParamOutDriver.siModOfOpt_6060 AT %QB."Traverser".ModesOfOperation_6060;
	::Trav:tyParamInDriver.siModOfOptDisp_6061 AT %IB."Traverser".ModesOfOperationDisplay_6061;
	::Trav:tyParamInDriver.diActualPos_6064 AT %ID."Traverser".PositionActualValue_6064;
	::Trav:tyParamOutDriver.diTargetPos_607A AT %QD."Traverser".TargetPosition_607A;
	::Trav:tyParamOutDriver.udiMoveSpd_6081 AT %QD."Traverser".ProfileVelocity_6081;
	::Trav:tyParamOutDriver.siHmMethod_6098 AT %QB."Traverser".HomingMethod_6098;
	::Trav:tyParamInDriver.udiDigitalInputs_60FD AT %ID."Traverser".DigitalInputs_60FD;
	::Trav:tyParamOutDriver.diJogVel_60FF AT %QD."Traverser".TargetVelocity_60FF;
	::DOutput:a_bPhysicalDO[13] AT %QX."X20DO9321_X11".DigitalOutput07;
	::DOutput:a_bPhysicalDO[14] AT %QX."X20DO9321_X11".DigitalOutput08;
	::DOutput:a_bPhysicalDO[15] AT %QX."X20DO9321_X11".DigitalOutput09;
	::DOutput:a_bPhysicalDO[16] AT %QX."X20DO9321_X11".DigitalOutput10;
	::DOutput:a_bPhysicalDO[17] AT %QX."X20DO9321_X11".DigitalOutput11;
	::DOutput:a_bPhysicalDO[18] AT %QX."X20DO9321_X11".DigitalOutput12;
	::DInput:a_bPhysicalDI[61] AT %IX."X20DI9372_X7".DigitalInput01;
	::DInput:a_bPhysicalDI[62] AT %IX."X20DI9372_X7".DigitalInput02;
	::DInput:a_bPhysicalDI[63] AT %IX."X20DI9372_X7".DigitalInput03;
	::DInput:a_bPhysicalDI[64] AT %IX."X20DI9372_X7".DigitalInput04;
	::DInput:a_bPhysicalDI[65] AT %IX."X20DI9372_X7".DigitalInput05;
	::DInput:a_bPhysicalDI[66] AT %IX."X20DI9372_X7".DigitalInput06;
	::DOutput:a_bPhysicalDO[31] AT %QX."X20DO9321_X13".DigitalOutput01;
	::DOutput:a_bPhysicalDO[32] AT %QX."X20DO9321_X13".DigitalOutput02;
	::DOutput:a_bPhysicalDO[33] AT %QX."X20DO9321_X13".DigitalOutput03;
	::DOutput:a_bPhysicalDO[34] AT %QX."X20DO9321_X13".DigitalOutput04;
	::DOutput:a_bPhysicalDO[35] AT %QX."X20DO9321_X13".DigitalOutput05;
	::DOutput:a_bPhysicalDO[36] AT %QX."X20DO9321_X13".DigitalOutput06;
	::DOutput:a_bPhysicalDO[37] AT %QX."X20DO9321_X13".DigitalOutput07;
	::DOutput:a_bPhysicalDO[38] AT %QX."X20DO9321_X13".DigitalOutput08;
	::DOutput:a_bPhysicalDO[39] AT %QX."X20DO9321_X13".DigitalOutput09;
	::DOutput:a_bPhysicalDO[40] AT %QX."X20DO9321_X13".DigitalOutput10;
	::DOutput:a_bPhysicalDO[41] AT %QX."X20DO9321_X13".DigitalOutput11;
	::DOutput:a_bPhysicalDO[42] AT %QX."X20DO9321_X13".DigitalOutput12;
	::AWOpen:tyParamInDriver.uiErrCode_603F AT %IW."AutoWidth".Error_code_603F;
	::AWOpen:tyParamInDriver.siModOfOptDisp_6061 AT %IB."AutoWidth".Modes_of_operation_display_6061;
	::AWOpen:tyParamInDriver.diActualPos_6064 AT %ID."AutoWidth".Position_actual_value_6064;
	::AWOpen:tyParamInDriver.udiDigitalInputs_60FD AT %ID."AutoWidth".Digital_intputs_60FD;
	::AWOpen:tyParamOutDriver.siModOfOpt_6060 AT %QB."AutoWidth".Modes_of_operation_6060;
	::AWOpen:tyParamOutDriver.diTargetPos_607A AT %QD."AutoWidth".Target_position_607A;
	::AWOpen:tyParamOutDriver.udiMoveSpd_6081 AT %QD."AutoWidth".Profile_velocity_6081;
	::AWOpen:tyParamOutDriver.siHmMethod_6098 AT %QB."AutoWidth".Homing_method_6098;
	::AWOpen:tyParamOutDriver.diJogVel_60FF AT %QD."AutoWidth".Target_velocity_60FF;
	::LifterBtm:tyParamOutDriver.siModOfOpt_6060 AT %QB."Lifter".Modes_of_operation_6060;
	::LifterBtm:tyParamOutDriver.diTargetPos_607A AT %QD."Lifter".Target_position_607A;
	::LifterBtm:tyParamOutDriver.udiMoveSpd_6081 AT %QD."Lifter".Profile_velocity_6081;
	::LifterBtm:tyParamOutDriver.siHmMethod_6098 AT %QB."Lifter".Homing_method_6098;
	::LifterBtm:tyParamOutDriver.diJogVel_60FF AT %QD."Lifter".Target_velocity_60FF;
	::LifterBtm:tyParamInDriver.uiErrCode_603F AT %IW."Lifter".Error_code_603F;
	::LifterBtm:tyParamInDriver.siModOfOptDisp_6061 AT %IB."Lifter".Modes_of_operation_display_6061;
	::LifterBtm:tyParamInDriver.diActualPos_6064 AT %ID."Lifter".Position_actual_value_6064;
	::LifterBtm:tyParamInDriver.udiDigitalInputs_60FD AT %ID."Lifter".Digital_intputs_60FD;
	::Trav:tyParamOutDriver.siModOfOpt_6060 AT %QB."Traverser".Modes_of_operation_6060;
	::Trav:tyParamOutDriver.diTargetPos_607A AT %QD."Traverser".Target_position_607A;
	::Trav:tyParamOutDriver.udiMoveSpd_6081 AT %QD."Traverser".Profile_velocity_6081;
	::Trav:tyParamOutDriver.siHmMethod_6098 AT %QB."Traverser".Homing_method_6098;
	::Trav:tyParamOutDriver.diJogVel_60FF AT %QD."Traverser".Target_velocity_60FF;
	::Trav:tyParamInDriver.uiErrCode_603F AT %IW."Traverser".Error_code_603F;
	::Trav:tyParamInDriver.siModOfOptDisp_6061 AT %IB."Traverser".Modes_of_operation_display_6061;
	::Trav:tyParamInDriver.diActualPos_6064 AT %ID."Traverser".Position_actual_value_6064;
	::Trav:tyParamInDriver.udiDigitalInputs_60FD AT %ID."Traverser".Digital_intputs_60FD;
	::AWPushOrPu:bModuleOK AT %IX."PullerAutoWidth".ModuleOk;
	::AWPushOrPu:tyParamInDriver.uiErrCode_603F AT %IW."PullerAutoWidth".Error_code_603F;
	::AWPushOrPu:tyParamOutDriver.uiCtrlword_6040 AT %QW."PullerAutoWidth".Controlword_6040;
	::AWPushOrPu:tyParamInDriver.uiStatword_6041 AT %IW."PullerAutoWidth".Statusword_6041;
	::AWPushOrPu:tyParamInDriver.siModOfOptDisp_6061 AT %IB."PullerAutoWidth".Modes_of_operation_display_6061;
	::AWPushOrPu:tyParamInDriver.diActualPos_6064 AT %ID."PullerAutoWidth".Position_actual_value_6064;
	::AWPushOrPu:tyParamInDriver.udiDigitalInputs_60FD AT %ID."PullerAutoWidth".Digital_intputs_60FD;
	::AWPushOrPu:tyParamOutDriver.siModOfOpt_6060 AT %QB."PullerAutoWidth".Modes_of_operation_6060;
	::AWPushOrPu:tyParamOutDriver.diTargetPos_607A AT %QD."PullerAutoWidth".Target_position_607A;
	::AWPushOrPu:tyParamOutDriver.udiMoveSpd_6081 AT %QD."PullerAutoWidth".Profile_velocity_6081;
	::AWPushOrPu:tyParamOutDriver.siHmMethod_6098 AT %QB."PullerAutoWidth".Homing_method_6098;
	::AWPushOrPu:tyParamOutDriver.diJogVel_60FF AT %QD."PullerAutoWidth".Target_velocity_60FF;
	::DInput:a_bPhysicalDI[37] AT %IX."X20DI9372_X5".DigitalInput01;
	::DInput:a_bPhysicalDI[38] AT %IX."X20DI9372_X5".DigitalInput02;
	::DInput:a_bPhysicalDI[39] AT %IX."X20DI9372_X5".DigitalInput03;
	::DInput:a_bPhysicalDI[40] AT %IX."X20DI9372_X5".DigitalInput04;
	::DInput:a_bPhysicalDI[41] AT %IX."X20DI9372_X5".DigitalInput05;
	::DInput:a_bPhysicalDI[42] AT %IX."X20DI9372_X5".DigitalInput06;
	::DInput:a_bPhysicalDI[43] AT %IX."X20DI9372_X5".DigitalInput07;
	::DInput:a_bPhysicalDI[44] AT %IX."X20DI9372_X5".DigitalInput08;
	::DInput:a_bPhysicalDI[45] AT %IX."X20DI9372_X5".DigitalInput09;
	::DInput:a_bPhysicalDI[46] AT %IX."X20DI9372_X5".DigitalInput10;
	::DInput:a_bPhysicalDI[47] AT %IX."X20DI9372_X5".DigitalInput11;
	::DInput:a_bPhysicalDI[48] AT %IX."X20DI9372_X5".DigitalInput12;
	::DInput:a_bPhysicalDI[49] AT %IX."X20DI9372_X6".DigitalInput01;
	::DInput:a_bPhysicalDI[50] AT %IX."X20DI9372_X6".DigitalInput02;
	::DInput:a_bPhysicalDI[51] AT %IX."X20DI9372_X6".DigitalInput03;
	::DInput:a_bPhysicalDI[52] AT %IX."X20DI9372_X6".DigitalInput04;
	::DInput:a_bPhysicalDI[53] AT %IX."X20DI9372_X6".DigitalInput05;
	::DInput:a_bPhysicalDI[54] AT %IX."X20DI9372_X6".DigitalInput06;
	::DInput:a_bPhysicalDI[55] AT %IX."X20DI9372_X6".DigitalInput07;
	::DInput:a_bPhysicalDI[56] AT %IX."X20DI9372_X6".DigitalInput08;
	::DInput:a_bPhysicalDI[57] AT %IX."X20DI9372_X6".DigitalInput09;
	::DInput:a_bPhysicalDI[58] AT %IX."X20DI9372_X6".DigitalInput10;
	::DInput:a_bPhysicalDI[59] AT %IX."X20DI9372_X6".DigitalInput11;
	::DInput:a_bPhysicalDI[60] AT %IX."X20DI9372_X6".DigitalInput12;
	::DOutput:a_bPhysicalDO[1] AT %QX."X20DO6321_X11".DigitalOutput01;
	::DOutput:a_bPhysicalDO[2] AT %QX."X20DO6321_X11".DigitalOutput02;
	::DOutput:a_bPhysicalDO[3] AT %QX."X20DO6321_X11".DigitalOutput03;
	::DOutput:a_bPhysicalDO[4] AT %QX."X20DO6321_X11".DigitalOutput04;
	::DOutput:a_bPhysicalDO[5] AT %QX."X20DO6321_X11".DigitalOutput05;
	::DOutput:a_bPhysicalDO[6] AT %QX."X20DO6321_X11".DigitalOutput06;
	::DOutput:a_bPhysicalDO[19] AT %QX."X20DO9321_X12".DigitalOutput01;
	::DOutput:a_bPhysicalDO[20] AT %QX."X20DO9321_X12".DigitalOutput02;
	::DOutput:a_bPhysicalDO[21] AT %QX."X20DO9321_X12".DigitalOutput03;
	::DOutput:a_bPhysicalDO[22] AT %QX."X20DO9321_X12".DigitalOutput04;
	::DOutput:a_bPhysicalDO[23] AT %QX."X20DO9321_X12".DigitalOutput05;
	::DOutput:a_bPhysicalDO[24] AT %QX."X20DO9321_X12".DigitalOutput06;
	::DOutput:a_bPhysicalDO[25] AT %QX."X20DO9321_X12".DigitalOutput07;
	::DOutput:a_bPhysicalDO[26] AT %QX."X20DO9321_X12".DigitalOutput08;
	::DOutput:a_bPhysicalDO[27] AT %QX."X20DO9321_X12".DigitalOutput09;
	::DOutput:a_bPhysicalDO[28] AT %QX."X20DO9321_X12".DigitalOutput10;
	::DOutput:a_bPhysicalDO[29] AT %QX."X20DO9321_X12".DigitalOutput11;
	::DOutput:a_bPhysicalDO[30] AT %QX."X20DO9321_X12".DigitalOutput12;
	::DOutput:a_bPhysicalDO[43] AT %QX."X20DO9321_X14".DigitalOutput01;
	::DOutput:a_bPhysicalDO[44] AT %QX."X20DO9321_X14".DigitalOutput02;
	::DOutput:a_bPhysicalDO[45] AT %QX."X20DO9321_X14".DigitalOutput03;
	::DOutput:a_bPhysicalDO[46] AT %QX."X20DO9321_X14".DigitalOutput04;
	::DOutput:a_bPhysicalDO[47] AT %QX."X20DO9321_X14".DigitalOutput05;
	::DOutput:a_bPhysicalDO[48] AT %QX."X20DO9321_X14".DigitalOutput06;
	::DOutput:a_bPhysicalDO[49] AT %QX."X20DO9321_X14".DigitalOutput07;
	::DOutput:a_bPhysicalDO[50] AT %QX."X20DO9321_X14".DigitalOutput08;
	::DOutput:a_bPhysicalDO[51] AT %QX."X20DO9321_X14".DigitalOutput09;
	::DOutput:a_bPhysicalDO[52] AT %QX."X20DO9321_X14".DigitalOutput10;
	::DOutput:a_bPhysicalDO[53] AT %QX."X20DO9321_X14".DigitalOutput11;
	::DOutput:a_bPhysicalDO[54] AT %QX."X20DO9321_X14".DigitalOutput12;
	::DOutput:a_bPhysicalDO[1] AT %QX."X20DO6321_X9".DigitalOutput01;
	::DOutput:a_bPhysicalDO[2] AT %QX."X20DO6321_X9".DigitalOutput02;
	::DOutput:a_bPhysicalDO[3] AT %QX."X20DO6321_X9".DigitalOutput03;
	::DOutput:a_bPhysicalDO[4] AT %QX."X20DO6321_X9".DigitalOutput04;
	::DOutput:a_bPhysicalDO[5] AT %QX."X20DO6321_X9".DigitalOutput05;
	::DOutput:a_bPhysicalDO[6] AT %QX."X20DO6321_X9".DigitalOutput06;
	::AWPushOrPu:tyParamInDriver.siModOfOptDisp_6061 AT %IB."PullerAutoWidth".ModesOfOperationDisplay_6061;
	::AWPushOrPu:tyParamInDriver.diActualPos_6064 AT %ID."PullerAutoWidth".PositionActualValue_6064;
	::AWPushOrPu:tyParamInDriver.udiDigitalInputs_60FD AT %ID."PullerAutoWidth".DigitalInputs_60FD;
	::AWPushOrPu:tyParamOutDriver.siModOfOpt_6060 AT %QB."PullerAutoWidth".ModesOfOperation_6060;
	::AWPushOrPu:tyParamOutDriver.diTargetPos_607A AT %QD."PullerAutoWidth".TargetPosition_607A;
	::AWPushOrPu:tyParamOutDriver.udiMoveSpd_6081 AT %QD."PullerAutoWidth".ProfileVelocity_6081;
	::AWPushOrPu:tyParamOutDriver.siHmMethod_6098 AT %QB."PullerAutoWidth".HomingMethod_6098;
	::AWPushOrPu:tyParamOutDriver.diJogVel_60FF AT %QD."PullerAutoWidth".TargetVelocity_60FF;
	::PullerPush:bModuleOK AT %IX."PullerPusher".ModuleOk;
	::PullerPush:tyParamInDriver.uiErrCode_603F AT %IW."PullerPusher".ErrorCode_603F;
	::PullerPush:tyParamInDriver.uiStatword_6041 AT %IW."PullerPusher".Statusword_6041;
	::PullerPush:tyParamInDriver.siModOfOptDisp_6061 AT %IB."PullerPusher".ModesOfOperationDisplay_6061;
	::PullerPush:tyParamInDriver.udiDigitalInputs_60FD AT %ID."PullerPusher".DigitalInputs_60FD;
	::PullerPush:tyParamOutDriver.uiCtrlword_6040 AT %QW."PullerPusher".Controlword_6040;
	::PullerPush:tyParamOutDriver.siModOfOpt_6060 AT %QB."PullerPusher".ModesOfOperation_6060;
	::PullerPush:tyParamInDriver.diActualPos_6064 AT %ID."PullerPusher".PositionActualValue_6064;
	::PullerPush:tyParamOutDriver.diTargetPos_607A AT %QD."PullerPusher".TargetPosition_607A;
	::PullerPush:tyParamOutDriver.udiMoveSpd_6081 AT %QD."PullerPusher".ProfileVelocity_6081;
	::PullerPush:tyParamOutDriver.siHmMethod_6098 AT %QB."PullerPusher".HomingMethod_6098;
	::PullerPush:tyParamOutDriver.diJogVel_60FF AT %QD."PullerPusher".TargetVelocity_60FF;
	::DInput:a_bPhysicalDI[67] AT %IX."X20DI9372_X7".DigitalInput07;
	::DInput:a_bPhysicalDI[68] AT %IX."X20DI9372_X7".DigitalInput08;
	::DInput:a_bPhysicalDI[69] AT %IX."X20DI9372_X7".DigitalInput09;
	::DInput:a_bPhysicalDI[70] AT %IX."X20DI9372_X7".DigitalInput10;
	::DInput:a_bPhysicalDI[71] AT %IX."X20DI9372_X7".DigitalInput11;
	::DInput:a_bPhysicalDI[72] AT %IX."X20DI9372_X7".DigitalInput12;
	::AWPushOrPu:tyParamInDriver.uiErrCode_603F AT %IW."PullerAutoWidth".ErrorCode_603F;
END_VAR
```

## Configuration 3Mag_RotMtrPuller_Estun

### Task classes (Cpu.sw)
```
Cyclic#1 (cycle 10000 us, tolerance 10000 us):
  DInput <- DInput.DInput.prg
  DOutput <- DOutput.DOutput.prg
Cyclic#2 (cycle 20000 us, tolerance 20000 us):
  BarcodeRdr <- USBBarcodeRdr.BarcodeRdr.prg
  PullConv <- Conv.PullConv.prg
  MagConv2Cl <- MagConv.MagConv2Clp1.prg
  MagConv2C1 <- MagConv.MagConv2Clp2.prg
  MagConv2C2 <- MagConv.MagConv2Clp3.prg
  MagConv2C3 <- MagConv.MagConv2Clp4.prg
  MtrPshr <- MtrPshr.MtrPshr.prg
Cyclic#3 (cycle 50000 us, tolerance 50000 us):
  UI <- UI.UI.prg
  Startup <- Startup.Startup.prg
  General <- General.General.prg
  UsrFolder <- UsrFolder.UsrFolder.prg
  LibVer <- LibVer.LibVer.prg
  Time <- Time.Time.prg
  HWInfo <- HWInfo.HWInfo.prg
  TLBuz <- TLBuz.TLBuz.prg
  Alarm <- Alarm.Alarm.prg
  RstErr <- RstErr.RstErr.prg
  ProdRcp <- ProdRcp.ProdRcp.prg
  MpProdRcp <- MpProdRcp.MpProdRcp.prg
  MagRcp <- MagRcp.MagRcp.prg
  MagRcp1 <- MagRcp.MagRcp1.prg
  McParam <- McParam.McParam.prg
  NtParam <- NtParam.NtParam.prg
  UsrMgmt <- UsrMgmt.UsrMgmt.prg
  Buffer1 <- Buffer.Buffer1.prg
  Buffer2 <- Buffer.Buffer2.prg
  Buffer3 <- Buffer.Buffer3.prg
  Buffer4 <- Buffer.Buffer4.prg
  USSMEMA1 <- SMEMA.USSMEMA1.prg
  USSMEMA2 <- SMEMA.USSMEMA2.prg
  USSMEMA3 <- SMEMA.USSMEMA3.prg
  USSMEMA4 <- SMEMA.USSMEMA4.prg
  DSSMEMA1 <- SMEMA.DSSMEMA1.prg
  DSSMEMA2 <- SMEMA.DSSMEMA2.prg
  DSSMEMA3 <- SMEMA.DSSMEMA3.prg
  DSSMEMA4 <- SMEMA.DSSMEMA4.prg
  DSSMEMAA <- SMEMA.DSSMEMAA.prg
  DSSMEMAB <- SMEMA.DSSMEMAB.prg
  Pneu2SenIn <- Pneu.Pneu2SenInShutter.prg
  Pneu2SenOu <- Pneu.Pneu2SenOutShutter.prg
  Pneu2SenPu <- Pneu.Pneu2SenPuller.prg
  Pneu2SenMa <- Pneu.MagSafetyBar.Pneu2SenMag1SafetyBar.prg
  Pneu2SenM1 <- Pneu.MagSafetyBar.Pneu2SenMag2SafetyBar.prg
  Pneu2SenM2 <- Pneu.MagSafetyBar.Pneu2SenMag3SafetyBar.prg
  Pneu2SenM3 <- Pneu.MagSafetyBar.Pneu2SenMag4SafetyBar.prg
  AWPushOrPu <- CANOpenServo.AW.AWPushOrPuller.prg
  AWOpen <- CANOpenServo.AW.AWOpen.prg
  Trav <- CANOpenServo.Trav.Trav.prg
  LifterBtm <- CANOpenServo.Lifter.LifterBtm.prg
  Hermes <- Hermes.Hermes.prg
  DSHermesA <- Hermes.DSHermesA.prg
  DSHermesB <- Hermes.DSHermesB.prg
  RmtHermes <- Hermes.RmtHermes.prg
  LFLeader <- LF.LFLeader.prg
  LFFollower <- LF.LFFollower.prg
  Follower1 <- LF.Follower1.prg
  Follower2 <- LF.Follower2.prg
  LCS <- LCS.LCS.prg
  LCSMngRcp <- LCS.LCSMngRcp.prg
  LCSLF <- LCS.LCSLF.prg
  Ops <- Operations.Ops.prg
  OpsTravLif <- Operations.OpsTravLifLD.prg
  OpsMagConv <- Operations.OpsMagConvLD1.prg
  OpsMagCon1 <- Operations.OpsMagConvLD2.prg
  OpsMagCon2 <- Operations.OpsMagConvLD3.prg
  OpsMagCon3 <- Operations.OpsMagConvLD4.prg
  OpsLifMagL <- Operations.OpsLifMagLD.prg
  AGV <- AGVCom.AGV.prg
  AGV1 <- AGVCom.AGV1.prg
  AGV2 <- AGVCom.AGV2.prg
  AGV3 <- AGVCom.AGV3.prg
  AGV4 <- AGVCom.AGV4.prg
  Pneu2SenSe <- Pneu.SelClamp.Pneu2SenSelClamp1.prg
  Pneu2SenS1 <- Pneu.SelClamp.Pneu2SenSelClamp2.prg
  Pneu2SenS2 <- Pneu.SelClamp.Pneu2SenSelClamp3.prg
  Pneu2SenS3 <- Pneu.SelClamp.Pneu2SenSelClamp4.prg
  Simu <- Simulation.Simu.prg
  USSOT1 <- SOT.USSOT1.prg
  DSSOT1 <- SOT.DSSOT1.prg
  USSOT2 <- SOT.USSOT2.prg
  DSSOT2 <- SOT.DSSOT2.prg
  USSOT3 <- SOT.USSOT3.prg
  DSSOT3 <- SOT.DSSOT3.prg
  USSOT4 <- SOT.USSOT4.prg
  DSSOT4 <- SOT.DSSOT4.prg
  Machine <- Machine.Machine.prg
  Machine1 <- Machine.Machine1.prg
  Frame <- RS232.DVFrame.Frame.prg
DataObjects: Acp10sys
VcDataObjects: Visu <- UI.Visu.dob
Binaries: vccdt, vccbmp, Visu03, vcfile, arial, vctcal, arialxsr, vcmgr, visvc, vccstr, vcbclass, vccbtn, vcgclass, vcdsint, vcnet, vccline, vcshared, vccddbox, arialbd, vccnum, vcpdvnc, vcpdsw, vccslider, vccbar, vcctext, Visu01, arialbi, vcfntttf, vccovl, vccshape, vcalarm, Visu02, vcrt, udbdef, vccpopup, vcdsloc, vcchspot, TCData, arsvcreg, vcpkat, vcpfgen, User, sysconf, ashwac, ashwd, Role, asfw, arconfig, iomap, Config, vcpfar00, acp10cfg, Acp10map, OpcUaMap
Libraries: standard, runtime, astime, asstring, operator, AsIecCon, AsCANopen, visapi, FileIO, AsIODiag, AsMem, dvframe, AsOpcUac, AsARCfg, sys_lib, AsTCP, MpRecipe, AsFltGen, brsystem, NtBuffer, NtConv, NtFileIO, NtLogFile, NtSMEMA, NtMem, NtMessage, NtOPCUA, NtOvenInfo, NtPneu, NtRS232, NtTLBuz, NtTCP, NtVersion, MpCom, MpBase, AsUSB, NtSOT, NtUSB, vcresman, dataobj, powerlnk, NtGeneral, NtUI
```

### Hardware
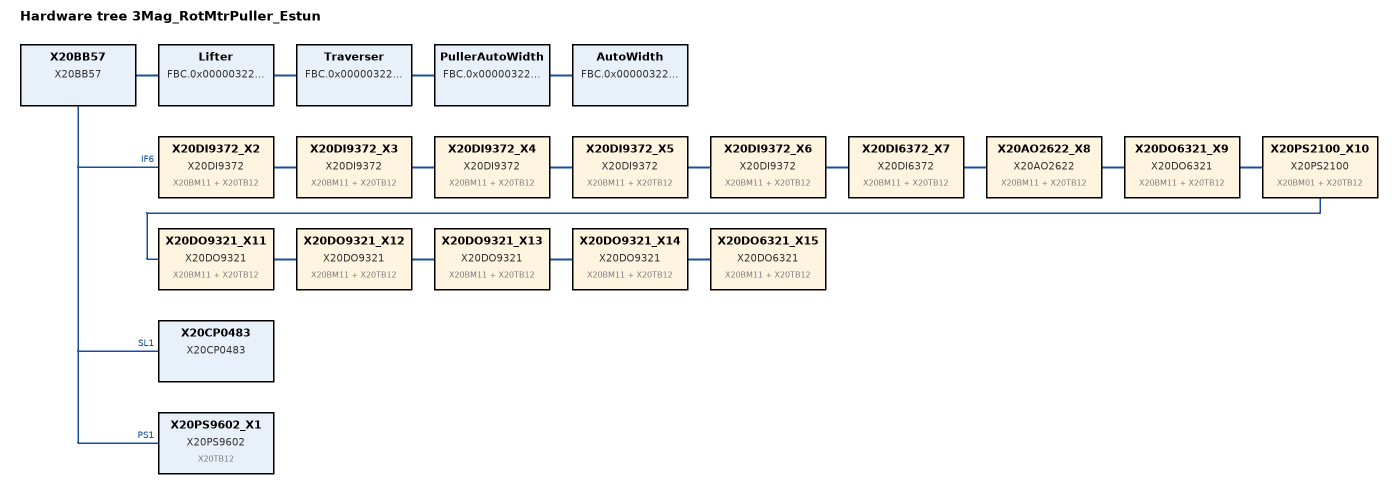
```
AutoWidth : FBC.0x00000322.0x00001000.NUTEK_ESTUN_PronetPlus_EDS_V106 v1.06.1 (OrderNumber=NUTEK_ESTUN_PronetPlus_V106)  [CAN1 -> PullerAutoWidth.CAN2 (NodeNumber=16)]
Lifter : FBC.0x00000322.0x00001000.NUTEK_ESTUN_PronetPlus_EDS_V106 v1.06.1 (OrderNumber=NUTEK_ESTUN_PronetPlus_V106)  [CAN1 -> X20BB57.IF7 (NodeNumber=17)]
PullerAutoWidth : FBC.0x00000322.0x00001000.NUTEK_ESTUN_PronetPlus_EDS_V106 v1.06.1 (OrderNumber=NUTEK_ESTUN_PronetPlus_V106)  [CAN1 -> Traverser.CAN2]
Traverser : FBC.0x00000322.0x00001000.NUTEK_ESTUN_PronetPlus_EDS_V106 v1.06.1 (OrderNumber=NUTEK_ESTUN_PronetPlus_V106)  [CAN1 -> Lifter.CAN2]
X20AO2622_X8 : X20AO2622 v1.2.0.0 (Disabled=true)  [SS1 -> X20TB12j.SS; SL -> X20BM11h.SL1]
X20BB57 : X20BB57 v1.1.1.0
  Connector IF1:
    Baudrate = 9600
    Parity = N
  Connector IF7:
    Baudrate = 1000000
    ActivateCanOpen = 1
    p100c_parametervalue = 1000
    p100d_parametervalue = 3
X20BM01 : X20BM01 v2.1.0.0 (Disabled=true)  [X2X1 -> X20BM11d.X2X2]
X20BM11 : X20BM11 v1.0.0.1 (Disabled=true)  [X2X1 -> X20BB57.IF6]
X20BM11a : X20BM11 v1.0.0.1 (Disabled=true)  [X2X1 -> X20BM11.X2X2]
X20BM11b : X20BM11 v1.0.0.1 (Disabled=true)  [X2X1 -> X20BM11a.X2X2]
X20BM11c : X20BM11 v1.0.0.1 (Disabled=true)  [X2X1 -> X20BM11e.X2X2]
X20BM11d : X20BM11 v1.0.0.1 (Disabled=true)  [X2X1 -> X20BM11h.X2X2]
X20BM11e : X20BM11 v1.0.0.1 (Disabled=true)  [X2X1 -> X20BM11f.X2X2]
X20BM11f : X20BM11 v1.0.0.1 (Disabled=true)  [X2X1 -> X20BM01.X2X2]
X20BM11g : X20BM11 v1.0.0.1 (Disabled=true)  [X2X1 -> X20BM11j.X2X2]
X20BM11h : X20BM11 v1.0.0.1 (Disabled=true)  [X2X1 -> X20BM11g.X2X2]
X20BM11i : X20BM11 v1.0.0.1 (Disabled=true)  [X2X1 -> X20BM11b.X2X2]
X20BM11j : X20BM11 v1.0.0.1 (Disabled=true)  [X2X1 -> X20BM11i.X2X2]
X20BM11k : X20BM11 v1.0.0.1 (Disabled=true)  [X2X1 -> X20BM11c.X2X2]
X20BM11n : X20BM11 v1.0.0.1 (Disabled=true)  [X2X1 -> X20BM11k.X2X2]
X20CP0483 : X20CP0483 v1.2.1.0  [SL -> X20BB57.SL1]
  Connector IF2:
    ActivateDevice = 1
    Mode = Manual
    InternetAddress = 192.168.0.2
    SubnetMask = 255.255.255.0
    Vnc1
    VncVcObjectName1 = Visu
    VncKeyMappingFile1 = VC\PS2-Keyboard.dis
    VncMaxConnections1 = 3
    VncRefreshRate1 = 100
    ActivateSnmp = 2
  ConfigurationID = NAELD003
  VolatileGlobalPvSize = 80000
  EnableUsbRemoteInstall = 1
  TimerDeviceType = SWIOTIMER
  Cyclic1Duration = 10000
  Cyclic1Tolerance = 10000
  Cyclic2Duration = 20000
  Cyclic2Tolerance = 20000
  Cyclic3Duration = 50000
  Cyclic3Tolerance = 50000
  Cyclic4Duration = 10000
  Cyclic4Tolerance = 10000
  Cyclic5Duration = 200000
  Cyclic5Tolerance = 200000
  Cyclic6Duration = 500000
  Cyclic6Tolerance = 500000
  Cyclic7Duration = 1000000
  Cyclic7Tolerance = 1000000
  Cyclic8Duration = 10000
  Cyclic8Tolerance = 10000
  FileDevice1
  FileDeviceName1 = C
  FileDevicePath1 = C:
  FileDevice2
  FileDeviceName2 = User
  FileDevicePath2 = C:\User
  FileDevice3
  FileDeviceName3 = Private
  FileDevicePath3 = C:\Private
  FileDevice4
  FileDeviceName4 = CustomerUser
  FileDevicePath4 = C:\User\UserMgmt
  FileDevice5
  FileDeviceName5 = ProdRcp
  FileDevicePath5 = C:\User\ProductRecipe
  FileDevice6
  FileDeviceName6 = MagRcp
  FileDevicePath6 = C:\User\MagazineRecipe
  FileDevice7
  FileDeviceName7 = Alarm
  FileDevicePath7 = C:\User\Alarm
  FileDevice8
  FileDeviceName8 = McParam
  FileDevicePath8 = C:\User\MachineParameter
  FileDevice9
  FileDeviceName9 = NtParam
  FileDevicePath9 = C:\Private\NutekParameter
  FileDevice10
  FileDeviceName10 = LibVer
  FileDevicePath10 = C:\User\LibrariesVersion
  FileDevice11
  FileDeviceName11 = Retain
  FileDevicePath11 = C:\User\Retain
  FileDevice12
  FileDeviceName12 = Log
  FileDevicePath12 = C:\User\Log
  FileDevice13
  FileDeviceName13 = LCS
  FileDevicePath13 = C:\User\LCS
  FileDevice14
  FileDeviceName14 = MpProdRcp
  FileDevicePath14 = C:\User\ProductRecipeXml
  FileDevice15
  FileDeviceName15 = MpNtParam
  FileDevicePath15 = C:\Private\NutekParameterXml
  FileDevice16
  FileDeviceName16 = MagRcp1
  FileDevicePath16 = C:\User\MagazineRecipe1
  FileDevice17
  FileDeviceName17 = Serial
  FileDevicePath17 = C:\User\Serial
  FileDevice18
  FileDeviceName18 = USB
  FileDevicePath18 = C:\User\Serial\USB
  FileDevice19
  FileDeviceName19 = RS232
  FileDevicePath19 = C:\User\Serial\RS232
  FtpUser1
  FtpUsername1 = NTAFTP
  FtpUserPassword1 = JmcONQZEIGyG0Pt+VekJRbxmc4fxS8REPwlCJguEtEY=  // NTA4BH
  FtpUserSalt1 = smKszLJT
  FTPAccessRight1 = 0
  FTPdevice1 = ALL
  FtpUser2
  FtpUsername2 = admin
  FtpUserPassword2 = GulCMI/jV0v16Ew6MS+jrzqmTLk+NRkNo3Y+jAhzSzY=  // admin
  FtpUserSalt2 = robUzvv7
  FTPAccessRight2 = 0
  FTPMSPartition2 = SYSTEM
  FTPMSpath2 = User
  FtpUser3
  FtpUsername3 = LCS
  FtpUserPassword3 = 6XI8rzr3QlcLzq1fKGxRBMxxRW19t00F0QlEDJIXmLc=  // LCS
  FtpUserSalt3 = Xz6TWjSu
  FTPMSPartition3 = SYSTEM
  FTPMSpath3 = User\LCS
  ActivateOpcUa = 1
  OpcUa_ConversationSecurityPolicy_EnableBasic256Rsa256 = 0
  OpcUaInformationModels_PV_Version = 1
X20DI6372_X7 : X20DI6372 v1.1.0.0 (Disabled=true)  [SS1 -> X20TB12i.SS; SL -> X20BM11g.SL1]
X20DI9372_X2 : X20DI9372 v1.1.0.0 (Disabled=true)  [SS1 -> X20TB12a.SS; SL -> X20BM11.SL1]
X20DI9372_X3 : X20DI9372 v1.1.0.0 (Disabled=true)  [SS1 -> X20TB12b.SS; SL -> X20BM11a.SL1]
X20DI9372_X4 : X20DI9372 v1.1.0.0 (Disabled=true)  [SS1 -> X20TB12c.SS; SL -> X20BM11b.SL1]
X20DI9372_X5 : X20DI9372 v1.1.0.0 (Disabled=true)  [SS1 -> X20TB12k.SS; SL -> X20BM11i.SL1]
X20DI9372_X6 : X20DI9372 v1.1.0.0 (Disabled=true)  [SS1 -> X20TB12l.SS; SL -> X20BM11j.SL1]
X20DO6321_X15 : X20DO6321 v1.1.0.0 (Disabled=true)  [SS1 -> X20TB12p.SS; SL -> X20BM11n.SL1]
X20DO6321_X9 : X20DO6321 v1.1.0.0 (Disabled=true)  [SS1 -> X20TB12e.SS; SL -> X20BM11d.SL1]
X20DO9321_X11 : X20DO9321 v1.1.0.0 (Disabled=true)  [SS1 -> X20TB12h.SS; SL -> X20BM11f.SL1]
X20DO9321_X12 : X20DO9321 v1.1.0.0 (Disabled=true)  [SS1 -> X20TB12g.SS; SL -> X20BM11e.SL1]
X20DO9321_X13 : X20DO9321 v1.1.0.0 (Disabled=true)  [SS1 -> X20TB12d.SS; SL -> X20BM11c.SL1]
X20DO9321_X14 : X20DO9321 v1.1.0.0 (Disabled=true)  [SS1 -> X20TB12m.SS; SL -> X20BM11k.SL1]
X20PS2100_X10 : X20PS2100 v1.2.0.0 (Disabled=true)  [SS1 -> X20TB12f.SS; SL -> X20BM01.SL1]
X20PS9602_X1 : X20PS9602 v1.0.2.0  [PS -> X20BB57.PS1; SS1 -> X20TB12.SS]
X20TB12 : X20TB12 v1.0.0.0
X20TB12a : X20TB12 v1.0.0.0 (Disabled=true)
X20TB12b : X20TB12 v1.0.0.0 (Disabled=true)
X20TB12c : X20TB12 v1.0.0.0 (Disabled=true)
X20TB12d : X20TB12 v1.0.0.0 (Disabled=true)
X20TB12e : X20TB12 v1.0.0.0 (Disabled=true)
X20TB12f : X20TB12 v1.0.0.0 (Disabled=true)
X20TB12g : X20TB12 v1.0.0.0 (Disabled=true)
X20TB12h : X20TB12 v1.0.0.0 (Disabled=true)
X20TB12i : X20TB12 v1.0.0.0 (Disabled=true)
X20TB12j : X20TB12 v1.0.0.0 (Disabled=true)
X20TB12k : X20TB12 v1.0.0.0 (Disabled=true)
X20TB12l : X20TB12 v1.0.0.0 (Disabled=true)
X20TB12m : X20TB12 v1.0.0.0 (Disabled=true)
X20TB12p : X20TB12 v1.0.0.0 (Disabled=true)
```
